  MoveL 2029 to (241.29, 57.14, 41.04) mm, rotated rx 180 ry 0 rz 180 deg; joints [-19.819, 17.595, 47.827, 40.909, 31.181, -36.55]
  Call Extruder(249.57521)
  MoveL 2030 to (241.29, 142.86, 41.03) mm, rotated rx 180 ry 0 rz 180 deg; joints [-28.232, 26.406, 35.284, 48.547, 39.135, -41.289]
  Call Extruder(250.00364)
  MoveL 2031 to (241.27, 143.74, 41.03) mm, rotated rx 180 ry 0 rz -180 deg; joints [-28.313, 26.529, 35.098, 48.584, 39.23, -41.288]
  MoveL 2032 to (241.27, 143.74, 41.03) mm, rotated rx 180 ry 0 rz -180 deg; joints [-28.313, 26.529, 35.098, 48.584, 39.23, -41.288]
  Call Extruder(250.57709)
  MoveL 2033 to (241.22, 144.9, 41.03) mm, rotated rx -180 ry 0 rz 180 deg; joints [-28.421, 26.688, 34.856, 48.637, 39.357, -41.289]
  MoveL 2034 to (241.22, 144.9, 41.03) mm, rotated rx -180 ry 0 rz 180 deg; joints [-28.421, 26.688, 34.856, 48.637, 39.357, -41.289]
  Call Extruder(251.01142)
  MoveL 2035 to (241.18, 145.77, 41.03) mm, rotated rx -180 ry 0 rz 180 deg; joints [-28.503, 26.806, 34.676, 48.678, 39.452, -41.291]
  MoveL 2036 to (241.18, 145.77, 41.03) mm, rotated rx -180 ry 0 rz 180 deg; joints [-28.503, 26.806, 34.676, 48.678, 39.452, -41.291]
  Call Extruder(251.30553)
  MoveL 2037 to (241.13, 146.36, 41.04) mm, rotated rx 180 ry 0 rz 180 deg; joints [-28.559, 26.882, 34.56, 48.708, 39.515, -41.295]
  MoveL 2038 to (241.13, 146.36, 41.04) mm, rotated rx 180 ry 0 rz 180 deg; joints [-28.559, 26.882, 34.56, 48.708, 39.515, -41.295]
  Call Extruder(251.60097)
  MoveL 2039 to (241.09, 146.95, 41.03) mm, rotated rx 180 ry 0 rz 180 deg; joints [-28.615, 26.958, 34.443, 48.737, 39.579, -41.298]
  MoveL 2040 to (241.09, 146.95, 41.03) mm, rotated rx 180 ry 0 rz 180 deg; joints [-28.615, 26.958, 34.443, 48.737, 39.579, -41.298]
  Call Extruder(251.84723)
  MoveL 2041 to (241.04, 147.44, 41.04) mm, rotated rx 180 ry 0 rz -180 deg; joints [-28.662, 27.019, 34.349, 48.762, 39.631, -41.302]
  MoveL 2042 to (241.04, 147.44, 41.04) mm, rotated rx 180 ry 0 rz -180 deg; joints [-28.662, 27.019, 34.349, 48.762, 39.631, -41.302]
  Call Extruder(252.04393)
  MoveL 2043 to (240.99, 147.83, 41.04) mm, rotated rx -180 ry 0 rz 180 deg; joints [-28.7, 27.066, 34.278, 48.784, 39.672, -41.307]
  MoveL 2044 to (240.99, 147.83, 41.04) mm, rotated rx -180 ry 0 rz 180 deg; joints [-28.7, 27.066, 34.278, 48.784, 39.672, -41.307]
  Call Extruder(252.24151)
  MoveL 2045 to (240.95, 148.22, 41.03) mm, rotated rx 180 ry 0 rz 180 deg; joints [-28.737, 27.112, 34.207, 48.806, 39.713, -41.312]
  MoveL 2046 to (240.95, 148.22, 41.03) mm, rotated rx 180 ry 0 rz 180 deg; joints [-28.737, 27.112, 34.207, 48.806, 39.713, -41.312]
  Call Extruder(252.43995)
  MoveL 2047 to (240.9, 148.6, 41.04) mm, rotated rx 180 ry 0 rz 180 deg; joints [-28.774, 27.159, 34.135, 48.827, 39.754, -41.316]
  MoveL 2048 to (240.9, 148.6, 41.04) mm, rotated rx 180 ry 0 rz 180 deg; joints [-28.774, 27.159, 34.135, 48.827, 39.754, -41.316]
  Call Extruder(252.63926)
  MoveL 2049 to (240.86, 148.99, 41.04) mm, rotated rx 180 ry 0 rz -180 deg; joints [-28.812, 27.206, 34.063, 48.848, 39.795, -41.32]
  MoveL 2050 to (240.86, 148.99, 41.04) mm, rotated rx 180 ry 0 rz -180 deg; joints [-28.812, 27.206, 34.063, 48.848, 39.795, -41.32]
  Call Extruder(252.79809)
  MoveL 2051 to (240.81, 149.3, 41.03) mm, rotated rx 180 ry 0 rz 180 deg; joints [-28.842, 27.24, 34.011, 48.867, 39.827, -41.326]
  MoveL 2052 to (240.81, 149.3, 41.03) mm, rotated rx 180 ry 0 rz 180 deg; joints [-28.842, 27.24, 34.011, 48.867, 39.827, -41.326]
  Call Extruder(252.95765)
  MoveL 2053 to (240.76, 149.6, 41.03) mm, rotated rx 180 ry 0 rz 180 deg; joints [-28.872, 27.274, 33.959, 48.886, 39.859, -41.332]
  MoveL 2054 to (240.76, 149.6, 41.03) mm, rotated rx 180 ry 0 rz 180 deg; joints [-28.872, 27.274, 33.959, 48.886, 39.859, -41.332]
  Call Extruder(253.11794)
  MoveL 2055 to (240.71, 149.91, 41.03) mm, rotated rx 180 ry 0 rz 180 deg; joints [-28.902, 27.308, 33.907, 48.905, 39.891, -41.338]
  MoveL 2056 to (240.71, 149.91, 41.03) mm, rotated rx 180 ry 0 rz 180 deg; joints [-28.902, 27.308, 33.907, 48.905, 39.891, -41.338]
  Call Extruder(253.27896)
  MoveL 2057 to (240.66, 150.21, 41.04) mm, rotated rx 180 ry 0 rz 180 deg; joints [-28.932, 27.342, 33.855, 48.924, 39.923, -41.343]
  MoveL 2058 to (240.66, 150.21, 41.04) mm, rotated rx 180 ry 0 rz 180 deg; joints [-28.932, 27.342, 33.855, 48.924, 39.923, -41.343]
  Call Extruder(253.44070)
  MoveL 2059 to (240.61, 150.52, 41.04) mm, rotated rx 180 ry 0 rz -180 deg; joints [-28.962, 27.376, 33.802, 48.942, 39.955, -41.348]
  MoveL 2060 to (240.61, 150.52, 41.04) mm, rotated rx 180 ry 0 rz -180 deg; joints [-28.962, 27.376, 33.802, 48.942, 39.955, -41.348]
  Call Extruder(253.60317)
  MoveL 2061 to (240.57, 150.83, 41.04) mm, rotated rx 180 ry 0 rz 180 deg; joints [-28.993, 27.411, 33.749, 48.961, 39.987, -41.354]
  MoveL 2062 to (240.57, 150.83, 41.04) mm, rotated rx 180 ry 0 rz 180 deg; joints [-28.993, 27.411, 33.749, 48.961, 39.987, -41.354]
  Call Extruder(253.73710)
  MoveL 2063 to (240.52, 151.08, 41.03) mm, rotated rx -180 ry 0 rz 180 deg; joints [-29.017, 27.436, 33.71, 48.977, 40.012, -41.36]
  MoveL 2064 to (240.52, 151.08, 41.03) mm, rotated rx -180 ry 0 rz 180 deg; joints [-29.017, 27.436, 33.71, 48.977, 40.012, -41.36]
  Call Extruder(253.87164)
  MoveL 2065 to (240.47, 151.32, 41.04) mm, rotated rx 180 ry 0 rz 180 deg; joints [-29.043, 27.461, 33.671, 48.994, 40.038, -41.366]
  MoveL 2066 to (240.47, 151.32, 41.04) mm, rotated rx 180 ry 0 rz 180 deg; joints [-29.043, 27.461, 33.671, 48.994, 40.038, -41.366]
  Call Extruder(254.00678)
  MoveL 2067 to (240.42, 151.57, 41.04) mm, rotated rx -180 ry 0 rz -180 deg; joints [-29.067, 27.486, 33.632, 49.011, 40.063, -41.373]
  MoveL 2068 to (240.42, 151.57, 41.04) mm, rotated rx -180 ry 0 rz -180 deg; joints [-29.067, 27.486, 33.632, 49.011, 40.063, -41.373]
  Call Extruder(254.14254)
  MoveL 2069 to (240.37, 151.82, 41.03) mm, rotated rx 180 ry 0 rz 180 deg; joints [-29.092, 27.512, 33.593, 49.028, 40.089, -41.379]
  MoveL 2070 to (240.37, 151.82, 41.03) mm, rotated rx 180 ry 0 rz 180 deg; joints [-29.092, 27.512, 33.593, 49.028, 40.089, -41.379]
  Call Extruder(254.27891)
  MoveL 2071 to (240.32, 152.07, 41.04) mm, rotated rx -180 ry 0 rz 180 deg; joints [-29.117, 27.537, 33.554, 49.045, 40.114, -41.385]
  MoveL 2072 to (240.32, 152.07, 41.04) mm, rotated rx -180 ry 0 rz 180 deg; joints [-29.117, 27.537, 33.554, 49.045, 40.114, -41.385]
  Call Extruder(254.41589)
  MoveL 2073 to (240.27, 152.32, 41.04) mm, rotated rx 180 ry 0 rz 180 deg; joints [-29.142, 27.563, 33.514, 49.061, 40.14, -41.391]
  MoveL 2074 to (240.27, 152.32, 41.04) mm, rotated rx 180 ry 0 rz 180 deg; joints [-29.142, 27.563, 33.514, 49.061, 40.14, -41.391]
  Call Extruder(254.55347)
  MoveL 2075 to (240.22, 152.57, 41.03) mm, rotated rx -180 ry 0 rz 180 deg; joints [-29.167, 27.589, 33.474, 49.078, 40.166, -41.396]
  MoveL 2076 to (240.22, 152.57, 41.03) mm, rotated rx -180 ry 0 rz 180 deg; joints [-29.167, 27.589, 33.474, 49.078, 40.166, -41.396]
  Call Extruder(254.66717)
  MoveL 2077 to (240.17, 152.77, 41.04) mm, rotated rx 180 ry 0 rz 180 deg; joints [-29.188, 27.609, 33.443, 49.092, 40.187, -41.402]
  MoveL 2078 to (240.17, 152.77, 41.04) mm, rotated rx 180 ry 0 rz 180 deg; joints [-29.188, 27.609, 33.443, 49.092, 40.187, -41.402]
  Call Extruder(254.78132)
  MoveL 2079 to (240.13, 152.98, 41.04) mm, rotated rx -180 ry 0 rz 180 deg; joints [-29.209, 27.629, 33.413, 49.106, 40.207, -41.408]
  MoveL 2080 to (240.13, 152.98, 41.04) mm, rotated rx -180 ry 0 rz 180 deg; joints [-29.209, 27.629, 33.413, 49.106, 40.207, -41.408]
  Call Extruder(254.89592)
  MoveL 2081 to (240.08, 153.18, 41.03) mm, rotated rx -180 ry 0 rz -180 deg; joints [-29.229, 27.649, 33.382, 49.121, 40.228, -41.413]
  MoveL 2082 to (240.08, 153.18, 41.03) mm, rotated rx -180 ry 0 rz -180 deg; joints [-29.229, 27.649, 33.382, 49.121, 40.228, -41.413]
  Call Extruder(255.01098)
  MoveL 2083 to (240.04, 153.39, 41.03) mm, rotated rx 180 ry 0 rz 180 deg; joints [-29.25, 27.669, 33.35, 49.135, 40.249, -41.419]
  MoveL 2084 to (240.04, 153.39, 41.03) mm, rotated rx 180 ry 0 rz 180 deg; joints [-29.25, 27.669, 33.35, 49.135, 40.249, -41.419]
  Call Extruder(255.13320)
  MoveL 2085 to (239.98, 153.6, 41.04) mm, rotated rx 180 ry 0 rz 180 deg; joints [-29.272, 27.687, 33.322, 49.151, 40.27, -41.426]
  MoveL 2086 to (239.98, 153.6, 41.04) mm, rotated rx 180 ry 0 rz 180 deg; joints [-29.272, 27.687, 33.322, 49.151, 40.27, -41.426]
  Call Extruder(255.26286)
  MoveL 2087 to (239.92, 153.82, 41.04) mm, rotated rx 180 ry 0 rz 180 deg; joints [-29.296, 27.704, 33.296, 49.171, 40.292, -41.437]
  MoveL 2088 to (239.92, 153.82, 41.04) mm, rotated rx 180 ry 0 rz 180 deg; joints [-29.296, 27.704, 33.296, 49.171, 40.292, -41.437]
  Call Extruder(255.39309)
  MoveL 2089 to (239.85, 154.05, 41.03) mm, rotated rx -180 ry 0 rz -180 deg; joints [-29.319, 27.72, 33.271, 49.19, 40.313, -41.447]
  MoveL 2090 to (239.85, 154.05, 41.03) mm, rotated rx -180 ry 0 rz -180 deg; joints [-29.319, 27.72, 33.271, 49.19, 40.313, -41.447]
  Call Extruder(255.52388)
  MoveL 2091 to (239.78, 154.27, 41.04) mm, rotated rx 180 ry 0 rz 180 deg; joints [-29.343, 27.737, 33.244, 49.209, 40.335, -41.457]
  MoveL 2092 to (239.78, 154.27, 41.04) mm, rotated rx 180 ry 0 rz 180 deg; joints [-29.343, 27.737, 33.244, 49.209, 40.335, -41.457]
  Call Extruder(255.65523)
  MoveL 2093 to (239.71, 154.5, 41.03) mm, rotated rx -180 ry 0 rz 180 deg; joints [-29.366, 27.754, 33.218, 49.228, 40.356, -41.467]
  MoveL 2094 to (239.71, 154.5, 41.03) mm, rotated rx -180 ry 0 rz 180 deg; joints [-29.366, 27.754, 33.218, 49.228, 40.356, -41.467]
  Call Extruder(255.76713)
  MoveL 2095 to (239.65, 154.68, 41.03) mm, rotated rx 180 ry 0 rz 180 deg; joints [-29.386, 27.767, 33.198, 49.245, 40.374, -41.476]
  MoveL 2096 to (239.65, 154.68, 41.03) mm, rotated rx 180 ry 0 rz 180 deg; joints [-29.386, 27.767, 33.198, 49.245, 40.374, -41.476]
  Call Extruder(255.87948)
  MoveL 2097 to (239.59, 154.87, 41.04) mm, rotated rx 180 ry 0 rz 180 deg; joints [-29.406, 27.78, 33.178, 49.261, 40.392, -41.485]
  MoveL 2098 to (239.59, 154.87, 41.04) mm, rotated rx 180 ry 0 rz 180 deg; joints [-29.406, 27.78, 33.178, 49.261, 40.392, -41.485]
  Call Extruder(255.99227)
  MoveL 2099 to (239.53, 155.06, 41.03) mm, rotated rx -180 ry 0 rz 180 deg; joints [-29.426, 27.793, 33.158, 49.278, 40.41, -41.495]
  MoveL 2100 to (239.53, 155.06, 41.03) mm, rotated rx -180 ry 0 rz 180 deg; joints [-29.426, 27.793, 33.158, 49.278, 40.41, -41.495]
  Call Extruder(256.10550)
  MoveL 2101 to (239.47, 155.25, 41.04) mm, rotated rx 180 ry 0 rz 180 deg; joints [-29.446, 27.806, 33.138, 49.295, 40.428, -41.504]
  MoveL 2102 to (239.47, 155.25, 41.04) mm, rotated rx 180 ry 0 rz 180 deg; joints [-29.446, 27.806, 33.138, 49.295, 40.428, -41.504]
  Call Extruder(256.21918)
  MoveL 2103 to (239.41, 155.44, 41.04) mm, rotated rx 180 ry 0 rz 180 deg; joints [-29.466, 27.82, 33.117, 49.312, 40.446, -41.513]
  MoveL 2104 to (239.41, 155.44, 41.04) mm, rotated rx 180 ry 0 rz 180 deg; joints [-29.466, 27.82, 33.117, 49.312, 40.446, -41.513]
  Call Extruder(256.40114)
  MoveL 2105 to (239.29, 155.73, 41.03) mm, rotated rx 180 ry 0 rz -180 deg; joints [-29.499, 27.832, 33.097, 49.343, 40.472, -41.533]
  MoveL 2106 to (239.29, 155.73, 41.03) mm, rotated rx 180 ry 0 rz -180 deg; joints [-29.499, 27.832, 33.097, 49.343, 40.472, -41.533]
  Call Extruder(256.58386)
  MoveL 2107 to (239.16, 156.02, 41.04) mm, rotated rx 180 ry 0 rz 180 deg; joints [-29.531, 27.845, 33.077, 49.374, 40.498, -41.553]
  MoveL 2108 to (239.16, 156.02, 41.04) mm, rotated rx 180 ry 0 rz 180 deg; joints [-29.531, 27.845, 33.077, 49.374, 40.498, -41.553]
  Call Extruder(256.75428)
  MoveL 2109 to (239.05, 156.29, 41.03) mm, rotated rx -180 ry 0 rz 180 deg; joints [-29.561, 27.857, 33.06, 49.403, 40.522, -41.572]
  MoveL 2110 to (239.05, 156.29, 41.03) mm, rotated rx -180 ry 0 rz 180 deg; joints [-29.561, 27.857, 33.06, 49.403, 40.522, -41.572]
  Call Extruder(256.91229)
  MoveL 2111 to (238.94, 156.54, 41.04) mm, rotated rx 180 ry 0 rz 180 deg; joints [-29.589, 27.867, 33.044, 49.43, 40.544, -41.59]
  MoveL 2112 to (238.94, 156.54, 41.04) mm, rotated rx 180 ry 0 rz 180 deg; joints [-29.589, 27.867, 33.044, 49.43, 40.544, -41.59]
  Call Extruder(257.07091)
  MoveL 2113 to (238.84, 156.79, 41.04) mm, rotated rx 180 ry 0 rz 180 deg; joints [-29.617, 27.877, 33.028, 49.457, 40.566, -41.608]
  MoveL 2114 to (238.84, 156.79, 41.04) mm, rotated rx 180 ry 0 rz 180 deg; joints [-29.617, 27.877, 33.028, 49.457, 40.566, -41.608]
  Call Extruder(257.27708)
  MoveL 2115 to (238.66, 157.09, 41.04) mm, rotated rx -180 ry 0 rz 180 deg; joints [-29.653, 27.876, 33.029, 49.499, 40.59, -41.64]
  MoveL 2116 to (238.66, 157.09, 41.04) mm, rotated rx -180 ry 0 rz 180 deg; joints [-29.653, 27.876, 33.029, 49.499, 40.59, -41.64]
  Call Extruder(257.48403)
  MoveL 2117 to (238.49, 157.4, 41.04) mm, rotated rx 180 ry 0 rz 180 deg; joints [-29.689, 27.875, 33.031, 49.541, 40.614, -41.672]
  MoveL 2118 to (238.49, 157.4, 41.04) mm, rotated rx 180 ry 0 rz 180 deg; joints [-29.689, 27.875, 33.031, 49.541, 40.614, -41.672]
  Call Extruder(257.69175)
  MoveL 2119 to (238.31, 157.7, 41.04) mm, rotated rx 180 ry 0 rz 180 deg; joints [-29.725, 27.875, 33.031, 49.582, 40.638, -41.704]
  MoveL 2120 to (238.31, 157.7, 41.04) mm, rotated rx 180 ry 0 rz 180 deg; joints [-29.725, 27.875, 33.031, 49.582, 40.638, -41.704]
  Call Extruder(257.90025)
  MoveL 2121 to (238.13, 158.01, 41.04) mm, rotated rx -180 ry 0 rz 180 deg; joints [-29.761, 27.874, 33.032, 49.624, 40.662, -41.736]
  MoveL 2122 to (238.13, 158.01, 41.04) mm, rotated rx -180 ry 0 rz 180 deg; joints [-29.761, 27.874, 33.032, 49.624, 40.662, -41.736]
  Call Extruder(258.07978)
  MoveL 2123 to (237.96, 158.25, 41.04) mm, rotated rx -180 ry 0 rz 180 deg; joints [-29.792, 27.864, 33.049, 49.665, 40.678, -41.769]
  MoveL 2124 to (237.96, 158.25, 41.04) mm, rotated rx -180 ry 0 rz 180 deg; joints [-29.792, 27.864, 33.049, 49.665, 40.678, -41.769]
  Call Extruder(258.41320)
  MoveL 2125 to (237.63, 158.7, 41.03) mm, rotated rx 180 ry 0 rz 180 deg; joints [-29.849, 27.844, 33.08, 49.74, 40.709, -41.832]
  MoveL 2126 to (237.63, 158.7, 41.03) mm, rotated rx 180 ry 0 rz 180 deg; joints [-29.849, 27.844, 33.08, 49.74, 40.709, -41.832]
  Call Extruder(258.74780)
  MoveL 2127 to (237.3, 159.15, 41.04) mm, rotated rx 180 ry 0 rz 180 deg; joints [-29.907, 27.824, 33.11, 49.815, 40.741, -41.894]
  Call Extruder(259.57575)
  MoveL 2128 to (236.39, 160.19, 41.03) mm, rotated rx 180 ry 0 rz 180 deg; joints [-30.046, 27.733, 33.251, 50.018, 40.802, -42.072]
  Call Extruder(260.40368)
  MoveL 2129 to (235.35, 161.1, 41.03) mm, rotated rx -180 ry 0 rz 180 deg; joints [-30.182, 27.588, 33.475, 50.241, 40.842, -42.281]
  Call Extruder(260.57099)
  MoveL 2130 to (235.13, 161.27, 41.04) mm, rotated rx 180 ry 0 rz 180 deg; joints [-30.208, 27.551, 33.532, 50.289, 40.847, -42.328]
  MoveL 2131 to (235.13, 161.27, 41.04) mm, rotated rx 180 ry 0 rz 180 deg; joints [-30.208, 27.551, 33.532, 50.289, 40.847, -42.328]
  Call Extruder(260.90442)
  MoveL 2132 to (234.68, 161.59, 41.04) mm, rotated rx 180 ry 0 rz -180 deg; joints [-30.261, 27.478, 33.646, 50.384, 40.857, -42.42]
  MoveL 2133 to (234.68, 161.59, 41.04) mm, rotated rx 180 ry 0 rz -180 deg; joints [-30.261, 27.478, 33.646, 50.384, 40.857, -42.42]
  Call Extruder(261.23666)
  MoveL 2134 to (234.23, 161.92, 41.04) mm, rotated rx 180 ry 0 rz 180 deg; joints [-30.314, 27.404, 33.758, 50.479, 40.868, -42.511]
  MoveL 2135 to (234.23, 161.92, 41.04) mm, rotated rx 180 ry 0 rz 180 deg; joints [-30.314, 27.404, 33.758, 50.479, 40.868, -42.511]
  Call Extruder(261.35431)
  MoveL 2136 to (234.05, 162.02, 41.04) mm, rotated rx -180 ry 0 rz 180 deg; joints [-30.331, 27.373, 33.807, 50.514, 40.869, -42.547]
  MoveL 2137 to (234.05, 162.02, 41.04) mm, rotated rx -180 ry 0 rz 180 deg; joints [-30.331, 27.373, 33.807, 50.514, 40.869, -42.547]
  Call Extruder(261.56204)
  MoveL 2138 to (233.75, 162.2, 41.04) mm, rotated rx -180 ry 0 rz 180 deg; joints [-30.363, 27.316, 33.894, 50.577, 40.871, -42.609]
  MoveL 2139 to (233.75, 162.2, 41.04) mm, rotated rx -180 ry 0 rz 180 deg; joints [-30.363, 27.316, 33.894, 50.577, 40.871, -42.609]
  Call Extruder(261.76899)
  MoveL 2140 to (233.45, 162.37, 41.04) mm, rotated rx -180 ry 0 rz 180 deg; joints [-30.394, 27.26, 33.98, 50.639, 40.873, -42.672]
  MoveL 2141 to (233.45, 162.37, 41.04) mm, rotated rx -180 ry 0 rz 180 deg; joints [-30.394, 27.26, 33.98, 50.639, 40.873, -42.672]
  Call Extruder(261.97516)
  MoveL 2142 to (233.14, 162.55, 41.03) mm, rotated rx 180 ry 0 rz 180 deg; joints [-30.426, 27.204, 34.066, 50.701, 40.875, -42.734]
  MoveL 2143 to (233.14, 162.55, 41.03) mm, rotated rx 180 ry 0 rz 180 deg; joints [-30.426, 27.204, 34.066, 50.701, 40.875, -42.734]
  Call Extruder(262.15683)
  MoveL 2144 to (232.87, 162.69, 41.04) mm, rotated rx 180 ry 0 rz 180 deg; joints [-30.453, 27.151, 34.148, 50.758, 40.876, -42.791]
  MoveL 2145 to (232.87, 162.69, 41.04) mm, rotated rx 180 ry 0 rz 180 deg; joints [-30.453, 27.151, 34.148, 50.758, 40.876, -42.791]
  Call Extruder(262.31480)
  MoveL 2146 to (232.62, 162.8, 41.04) mm, rotated rx 180 ry 0 rz 180 deg; joints [-30.476, 27.1, 34.227, 50.807, 40.874, -42.842]
  MoveL 2147 to (232.62, 162.8, 41.04) mm, rotated rx 180 ry 0 rz 180 deg; joints [-30.476, 27.1, 34.227, 50.807, 40.874, -42.842]
  Call Extruder(262.47217)
  MoveL 2148 to (232.37, 162.91, 41.04) mm, rotated rx 180 ry 0 rz 180 deg; joints [-30.498, 27.048, 34.305, 50.857, 40.872, -42.894]
  MoveL 2149 to (232.37, 162.91, 41.04) mm, rotated rx 180 ry 0 rz 180 deg; joints [-30.498, 27.048, 34.305, 50.857, 40.872, -42.894]
  Call Extruder(262.65491)
  MoveL 2150 to (232.07, 163.02, 41.04) mm, rotated rx -180 ry 0 rz 180 deg; joints [-30.524, 26.988, 34.398, 50.915, 40.869, -42.954]
  MoveL 2151 to (232.07, 163.02, 41.04) mm, rotated rx -180 ry 0 rz 180 deg; joints [-30.524, 26.988, 34.398, 50.915, 40.869, -42.954]
  Call Extruder(262.83690)
  MoveL 2152 to (231.78, 163.15, 41.03) mm, rotated rx -180 ry 0 rz 180 deg; joints [-30.551, 26.928, 34.49, 50.973, 40.867, -43.014]
  MoveL 2153 to (231.78, 163.15, 41.03) mm, rotated rx -180 ry 0 rz 180 deg; joints [-30.551, 26.928, 34.49, 50.973, 40.867, -43.014]
  Call Extruder(262.98424)
  MoveL 2154 to (231.54, 163.24, 41.04) mm, rotated rx 180 ry 0 rz 180 deg; joints [-30.571, 26.877, 34.567, 51.02, 40.865, -43.063]
  MoveL 2155 to (231.54, 163.24, 41.04) mm, rotated rx 180 ry 0 rz 180 deg; joints [-30.571, 26.877, 34.567, 51.02, 40.865, -43.063]
  Call Extruder(263.09746)
  MoveL 2156 to (231.35, 163.3, 41.03) mm, rotated rx 180 ry 0 rz 180 deg; joints [-30.587, 26.836, 34.63, 51.057, 40.861, -43.102]
  MoveL 2157 to (231.35, 163.3, 41.03) mm, rotated rx 180 ry 0 rz 180 deg; joints [-30.587, 26.836, 34.63, 51.057, 40.861, -43.102]
  Call Extruder(263.21024)
  MoveL 2158 to (231.17, 163.36, 41.03) mm, rotated rx 180 ry 0 rz 180 deg; joints [-30.602, 26.795, 34.693, 51.094, 40.858, -43.141]
  MoveL 2159 to (231.17, 163.36, 41.03) mm, rotated rx 180 ry 0 rz 180 deg; joints [-30.602, 26.795, 34.693, 51.094, 40.858, -43.141]
  Call Extruder(263.32257)
  MoveL 2160 to (230.98, 163.42, 41.04) mm, rotated rx 180 ry 0 rz 180 deg; joints [-30.618, 26.753, 34.756, 51.13, 40.855, -43.179]
  MoveL 2161 to (230.98, 163.42, 41.04) mm, rotated rx 180 ry 0 rz 180 deg; joints [-30.618, 26.753, 34.756, 51.13, 40.855, -43.179]
  Call Extruder(263.43446)
  MoveL 2162 to (230.79, 163.48, 41.04) mm, rotated rx 180 ry 0 rz 180 deg; joints [-30.633, 26.712, 34.818, 51.167, 40.852, -43.218]
  MoveL 2163 to (230.79, 163.48, 41.04) mm, rotated rx 180 ry 0 rz 180 deg; joints [-30.633, 26.712, 34.818, 51.167, 40.852, -43.218]
  Call Extruder(263.55586)
  MoveL 2164 to (230.58, 163.55, 41.04) mm, rotated rx 180 ry 0 rz 180 deg; joints [-30.65, 26.667, 34.887, 51.207, 40.849, -43.26]
  MoveL 2165 to (230.58, 163.55, 41.04) mm, rotated rx 180 ry 0 rz 180 deg; joints [-30.65, 26.667, 34.887, 51.207, 40.849, -43.26]
  Call Extruder(263.68667)
  MoveL 2166 to (230.36, 163.61, 41.03) mm, rotated rx -180 ry 0 rz 180 deg; joints [-30.668, 26.618, 34.962, 51.25, 40.845, -43.306]
  MoveL 2167 to (230.36, 163.61, 41.03) mm, rotated rx -180 ry 0 rz 180 deg; joints [-30.668, 26.618, 34.962, 51.25, 40.845, -43.306]
  Call Extruder(263.81692)
  MoveL 2168 to (230.14, 163.68, 41.03) mm, rotated rx 180 ry 0 rz 180 deg; joints [-30.685, 26.569, 35.036, 51.293, 40.842, -43.351]
  MoveL 2169 to (230.14, 163.68, 41.03) mm, rotated rx 180 ry 0 rz 180 deg; joints [-30.685, 26.569, 35.036, 51.293, 40.842, -43.351]
  Call Extruder(263.94661)
  MoveL 2170 to (229.91, 163.75, 41.04) mm, rotated rx 180 ry 0 rz 180 deg; joints [-30.703, 26.521, 35.11, 51.335, 40.838, -43.397]
  MoveL 2171 to (229.91, 163.75, 41.04) mm, rotated rx 180 ry 0 rz 180 deg; joints [-30.703, 26.521, 35.11, 51.335, 40.838, -43.397]
  Call Extruder(264.07572)
  MoveL 2172 to (229.69, 163.82, 41.03) mm, rotated rx -180 ry 0 rz 180 deg; joints [-30.721, 26.472, 35.185, 51.378, 40.834, -43.442]
  MoveL 2173 to (229.69, 163.82, 41.03) mm, rotated rx -180 ry 0 rz 180 deg; joints [-30.721, 26.472, 35.185, 51.378, 40.834, -43.442]
  Call Extruder(264.19080)
  MoveL 2174 to (229.48, 163.86, 41.04) mm, rotated rx 180 ry 0 rz 180 deg; joints [-30.736, 26.425, 35.256, 51.417, 40.83, -43.483]
  MoveL 2175 to (229.48, 163.86, 41.04) mm, rotated rx 180 ry 0 rz 180 deg; joints [-30.736, 26.425, 35.256, 51.417, 40.83, -43.483]
  Call Extruder(264.30542)
  MoveL 2176 to (229.28, 163.91, 41.04) mm, rotated rx 180 ry 0 rz 180 deg; joints [-30.751, 26.378, 35.327, 51.455, 40.825, -43.525]
  MoveL 2177 to (229.28, 163.91, 41.04) mm, rotated rx 180 ry 0 rz 180 deg; joints [-30.751, 26.378, 35.327, 51.455, 40.825, -43.525]
  Call Extruder(264.41959)
  MoveL 2178 to (229.08, 163.95, 41.04) mm, rotated rx 180 ry 0 rz -180 deg; joints [-30.766, 26.331, 35.398, 51.493, 40.82, -43.566]
  MoveL 2179 to (229.08, 163.95, 41.04) mm, rotated rx 180 ry 0 rz -180 deg; joints [-30.766, 26.331, 35.398, 51.493, 40.82, -43.566]
  Call Extruder(264.53331)
  MoveL 2180 to (228.87, 164, 41.03) mm, rotated rx 180 ry 0 rz 180 deg; joints [-30.781, 26.284, 35.468, 51.532, 40.815, -43.607]
  MoveL 2181 to (228.87, 164, 41.03) mm, rotated rx 180 ry 0 rz 180 deg; joints [-30.781, 26.284, 35.468, 51.532, 40.815, -43.607]
  Call Extruder(264.65873)
  MoveL 2182 to (228.65, 164.04, 41.03) mm, rotated rx 180 ry 0 rz 180 deg; joints [-30.797, 26.233, 35.547, 51.574, 40.81, -43.653]
  MoveL 2183 to (228.65, 164.04, 41.03) mm, rotated rx 180 ry 0 rz 180 deg; joints [-30.797, 26.233, 35.547, 51.574, 40.81, -43.653]
  Call Extruder(264.79570)
  MoveL 2184 to (228.4, 164.09, 41.04) mm, rotated rx 180 ry 0 rz -180 deg; joints [-30.815, 26.176, 35.633, 51.62, 40.804, -43.703]
  MoveL 2185 to (228.4, 164.09, 41.04) mm, rotated rx 180 ry 0 rz -180 deg; joints [-30.815, 26.176, 35.633, 51.62, 40.804, -43.703]
  Call Extruder(264.93207)
  MoveL 2186 to (228.15, 164.14, 41.04) mm, rotated rx 180 ry 0 rz 180 deg; joints [-30.832, 26.118, 35.72, 51.666, 40.798, -43.753]
  MoveL 2187 to (228.15, 164.14, 41.04) mm, rotated rx 180 ry 0 rz 180 deg; joints [-30.832, 26.118, 35.72, 51.666, 40.798, -43.753]
  Call Extruder(265.06783)
  MoveL 2188 to (227.9, 164.19, 41.04) mm, rotated rx 180 ry 0 rz -180 deg; joints [-30.85, 26.061, 35.806, 51.712, 40.792, -43.803]
  MoveL 2189 to (227.9, 164.19, 41.04) mm, rotated rx 180 ry 0 rz -180 deg; joints [-30.85, 26.061, 35.806, 51.712, 40.792, -43.803]
  Call Extruder(265.20298)
  MoveL 2190 to (227.65, 164.24, 41.03) mm, rotated rx 180 ry 0 rz 180 deg; joints [-30.868, 26.005, 35.891, 51.758, 40.787, -43.852]
  MoveL 2191 to (227.65, 164.24, 41.03) mm, rotated rx 180 ry 0 rz 180 deg; joints [-30.868, 26.005, 35.891, 51.758, 40.787, -43.852]
  Call Extruder(265.33751)
  MoveL 2192 to (227.4, 164.29, 41.04) mm, rotated rx 180 ry 0 rz 180 deg; joints [-30.886, 25.948, 35.977, 51.804, 40.781, -43.901]
  MoveL 2193 to (227.4, 164.29, 41.04) mm, rotated rx 180 ry 0 rz 180 deg; joints [-30.886, 25.948, 35.977, 51.804, 40.781, -43.901]
  Call Extruder(265.47144)
  MoveL 2194 to (227.15, 164.34, 41.04) mm, rotated rx -180 ry 0 rz -180 deg; joints [-30.903, 25.892, 36.061, 51.849, 40.776, -43.951]
  MoveL 2195 to (227.15, 164.34, 41.04) mm, rotated rx -180 ry 0 rz -180 deg; joints [-30.903, 25.892, 36.061, 51.849, 40.776, -43.951]
  Call Extruder(265.61931)
  MoveL 2196 to (226.87, 164.39, 41.03) mm, rotated rx -180 ry 0 rz 180 deg; joints [-30.923, 25.828, 36.157, 51.9, 40.769, -44.005]
  MoveL 2197 to (226.87, 164.39, 41.03) mm, rotated rx -180 ry 0 rz 180 deg; joints [-30.923, 25.828, 36.157, 51.9, 40.769, -44.005]
  Call Extruder(265.78105)
  MoveL 2198 to (226.57, 164.44, 41.04) mm, rotated rx 180 ry 0 rz 180 deg; joints [-30.943, 25.758, 36.263, 51.955, 40.762, -44.065]
  MoveL 2199 to (226.57, 164.44, 41.04) mm, rotated rx 180 ry 0 rz 180 deg; joints [-30.943, 25.758, 36.263, 51.955, 40.762, -44.065]
  Call Extruder(265.94206)
  MoveL 2200 to (226.26, 164.49, 41.04) mm, rotated rx 180 ry 0 rz 180 deg; joints [-30.964, 25.688, 36.368, 52.01, 40.755, -44.125]
  MoveL 2201 to (226.26, 164.49, 41.04) mm, rotated rx 180 ry 0 rz 180 deg; joints [-30.964, 25.688, 36.368, 52.01, 40.755, -44.125]
  Call Extruder(266.10234)
  MoveL 2202 to (225.96, 164.53, 41.03) mm, rotated rx -180 ry 0 rz 180 deg; joints [-30.985, 25.618, 36.473, 52.065, 40.748, -44.185]
  MoveL 2203 to (225.96, 164.53, 41.03) mm, rotated rx -180 ry 0 rz 180 deg; joints [-30.985, 25.618, 36.473, 52.065, 40.748, -44.185]
  Call Extruder(266.26190)
  MoveL 2204 to (225.65, 164.58, 41.04) mm, rotated rx 180 ry 0 rz 180 deg; joints [-31.006, 25.548, 36.578, 52.12, 40.741, -44.244]
  MoveL 2205 to (225.65, 164.58, 41.04) mm, rotated rx 180 ry 0 rz 180 deg; joints [-31.006, 25.548, 36.578, 52.12, 40.741, -44.244]
  Call Extruder(266.42073)
  MoveL 2206 to (225.34, 164.63, 41.03) mm, rotated rx 180 ry 0 rz -180 deg; joints [-31.027, 25.479, 36.682, 52.174, 40.734, -44.303]
  MoveL 2207 to (225.34, 164.63, 41.03) mm, rotated rx 180 ry 0 rz -180 deg; joints [-31.027, 25.479, 36.682, 52.174, 40.734, -44.303]
  Call Extruder(266.59940)
  MoveL 2208 to (225, 164.68, 41.04) mm, rotated rx 180 ry 0 rz -180 deg; joints [-31.049, 25.399, 36.801, 52.235, 40.726, -44.37]
  MoveL 2209 to (225, 164.68, 41.04) mm, rotated rx 180 ry 0 rz -180 deg; joints [-31.049, 25.399, 36.801, 52.235, 40.726, -44.37]
  Call Extruder(266.79784)
  MoveL 2210 to (224.61, 164.73, 41.04) mm, rotated rx -180 ry 0 rz -180 deg; joints [-31.074, 25.31, 36.934, 52.303, 40.716, -44.444]
  MoveL 2211 to (224.61, 164.73, 41.04) mm, rotated rx -180 ry 0 rz -180 deg; joints [-31.074, 25.31, 36.934, 52.303, 40.716, -44.444]
  Call Extruder(266.99542)
  MoveL 2212 to (224.22, 164.77, 41.03) mm, rotated rx 180 ry 0 rz 180 deg; joints [-31.1, 25.22, 37.067, 52.371, 40.707, -44.518]
  MoveL 2213 to (224.22, 164.77, 41.03) mm, rotated rx 180 ry 0 rz 180 deg; joints [-31.1, 25.22, 37.067, 52.371, 40.707, -44.518]
  Call Extruder(267.19212)
  MoveL 2214 to (223.84, 164.82, 41.04) mm, rotated rx 180 ry 0 rz 180 deg; joints [-31.125, 25.132, 37.199, 52.439, 40.698, -44.592]
  MoveL 2215 to (223.84, 164.82, 41.04) mm, rotated rx 180 ry 0 rz 180 deg; joints [-31.125, 25.132, 37.199, 52.439, 40.698, -44.592]
  Call Extruder(267.38796)
  MoveL 2216 to (223.45, 164.86, 41.03) mm, rotated rx 180 ry 0 rz 180 deg; joints [-31.15, 25.043, 37.331, 52.506, 40.69, -44.665]
  MoveL 2217 to (223.45, 164.86, 41.03) mm, rotated rx 180 ry 0 rz 180 deg; joints [-31.15, 25.043, 37.331, 52.506, 40.69, -44.665]
  Call Extruder(267.68332)
  MoveL 2218 to (222.86, 164.91, 41.04) mm, rotated rx 180 ry 0 rz 180 deg; joints [-31.186, 24.907, 37.534, 52.607, 40.675, -44.776]
  MoveL 2219 to (222.86, 164.91, 41.04) mm, rotated rx 180 ry 0 rz 180 deg; joints [-31.186, 24.907, 37.534, 52.607, 40.675, -44.776]
  Call Extruder(267.97734)
  MoveL 2220 to (222.27, 164.95, 41.04) mm, rotated rx 180 ry 0 rz 180 deg; joints [-31.222, 24.771, 37.736, 52.707, 40.66, -44.886]
  MoveL 2221 to (222.27, 164.95, 41.04) mm, rotated rx 180 ry 0 rz 180 deg; joints [-31.222, 24.771, 37.736, 52.707, 40.66, -44.886]
  Call Extruder(268.27004)
  MoveL 2222 to (221.68, 165, 41.04) mm, rotated rx 180 ry 0 rz 180 deg; joints [-31.258, 24.636, 37.935, 52.806, 40.647, -44.995]
  MoveL 2223 to (221.68, 165, 41.04) mm, rotated rx 180 ry 0 rz 180 deg; joints [-31.258, 24.636, 37.935, 52.806, 40.647, -44.995]
  Call Extruder(268.84349)
  MoveL 2224 to (220.52, 165.05, 41.04) mm, rotated rx 180 ry 0 rz 180 deg; joints [-31.326, 24.366, 38.334, 52.999, 40.617, -45.208]
  MoveL 2225 to (220.52, 165.05, 41.04) mm, rotated rx 180 ry 0 rz 180 deg; joints [-31.326, 24.366, 38.334, 52.999, 40.617, -45.208]
  Call Extruder(269.55750)
  MoveL 2226 to (219.06, 165.09, 41.03) mm, rotated rx 180 ry 0 rz 180 deg; joints [-31.409, 24.03, 38.827, 53.236, 40.582, -45.47]
  Call Extruder(386.40424)
  MoveL 2227 to (-19.06, 165.09, 41.04) mm, rotated rx 180 ry 0 rz 180 deg; joints [-51.475, -8.459, 76.118, 73.163, 54.823, -62.287]
  Call Extruder(386.83284)
  MoveL 2228 to (-19.94, 165.07, 41.04) mm, rotated rx -180 ry 0 rz 180 deg; joints [-51.582, -8.539, 76.186, 73.215, 54.921, -62.307]
  MoveL 2229 to (-19.94, 165.07, 41.04) mm, rotated rx -180 ry 0 rz 180 deg; joints [-51.582, -8.539, 76.186, 73.215, 54.921, -62.307]
  Call Extruder(387.40629)
  MoveL 2230 to (-21.1, 165.03, 41.04) mm, rotated rx 180 ry 0 rz 180 deg; joints [-51.722, -8.648, 76.277, 73.283, 55.051, -62.332]
  MoveL 2231 to (-21.1, 165.03, 41.04) mm, rotated rx 180 ry 0 rz 180 deg; joints [-51.722, -8.648, 76.277, 73.283, 55.051, -62.332]
  Call Extruder(387.84059)
  MoveL 2232 to (-21.97, 164.98, 41.04) mm, rotated rx 180 ry 0 rz 180 deg; joints [-51.827, -8.731, 76.347, 73.333, 55.147, -62.351]
  MoveL 2233 to (-21.97, 164.98, 41.04) mm, rotated rx 180 ry 0 rz 180 deg; joints [-51.827, -8.731, 76.347, 73.333, 55.147, -62.351]
  Call Extruder(388.13462)
  MoveL 2234 to (-22.56, 164.93, 41.04) mm, rotated rx 180 ry 0 rz -180 deg; joints [-51.897, -8.788, 76.395, 73.366, 55.212, -62.362]
  MoveL 2235 to (-22.56, 164.93, 41.04) mm, rotated rx 180 ry 0 rz -180 deg; joints [-51.897, -8.788, 76.395, 73.366, 55.212, -62.362]
  Call Extruder(388.42998)
  MoveL 2236 to (-23.15, 164.89, 41.04) mm, rotated rx 180 ry 0 rz 180 deg; joints [-51.966, -8.846, 76.443, 73.399, 55.276, -62.374]
  MoveL 2237 to (-23.15, 164.89, 41.04) mm, rotated rx 180 ry 0 rz 180 deg; joints [-51.966, -8.846, 76.443, 73.399, 55.276, -62.374]
  Call Extruder(388.67619)
  MoveL 2238 to (-23.64, 164.84, 41.04) mm, rotated rx 180 ry 0 rz 180 deg; joints [-52.023, -8.894, 76.483, 73.426, 55.328, -62.382]
  MoveL 2239 to (-23.64, 164.84, 41.04) mm, rotated rx 180 ry 0 rz 180 deg; joints [-52.023, -8.894, 76.483, 73.426, 55.328, -62.382]
  Call Extruder(388.87290)
  MoveL 2240 to (-24.03, 164.79, 41.04) mm, rotated rx -180 ry 0 rz 180 deg; joints [-52.067, -8.933, 76.516, 73.447, 55.37, -62.389]
  MoveL 2241 to (-24.03, 164.79, 41.04) mm, rotated rx -180 ry 0 rz 180 deg; joints [-52.067, -8.933, 76.516, 73.447, 55.37, -62.389]
  Call Extruder(389.07047)
  MoveL 2242 to (-24.42, 164.75, 41.04) mm, rotated rx 180 ry 0 rz 180 deg; joints [-52.112, -8.973, 76.548, 73.467, 55.411, -62.396]
  MoveL 2243 to (-24.42, 164.75, 41.04) mm, rotated rx 180 ry 0 rz 180 deg; joints [-52.112, -8.973, 76.548, 73.467, 55.411, -62.396]
  Call Extruder(389.26891)
  MoveL 2244 to (-24.8, 164.7, 41.04) mm, rotated rx 180 ry 0 rz 180 deg; joints [-52.156, -9.012, 76.581, 73.488, 55.452, -62.402]
  MoveL 2245 to (-24.8, 164.7, 41.04) mm, rotated rx 180 ry 0 rz 180 deg; joints [-52.156, -9.012, 76.581, 73.488, 55.452, -62.402]
  Call Extruder(389.46822)
  MoveL 2246 to (-25.19, 164.66, 41.04) mm, rotated rx 180 ry 0 rz 180 deg; joints [-52.2, -9.051, 76.614, 73.509, 55.493, -62.409]
  MoveL 2247 to (-25.19, 164.66, 41.04) mm, rotated rx 180 ry 0 rz 180 deg; joints [-52.2, -9.051, 76.614, 73.509, 55.493, -62.409]
  Call Extruder(389.62706)
  MoveL 2248 to (-25.5, 164.61, 41.04) mm, rotated rx -180 ry 0 rz 180 deg; joints [-52.235, -9.083, 76.64, 73.524, 55.525, -62.413]
  MoveL 2249 to (-25.5, 164.61, 41.04) mm, rotated rx -180 ry 0 rz 180 deg; joints [-52.235, -9.083, 76.64, 73.524, 55.525, -62.413]
  Call Extruder(389.78661)
  MoveL 2250 to (-25.8, 164.56, 41.04) mm, rotated rx -180 ry 0 rz 180 deg; joints [-52.269, -9.116, 76.667, 73.54, 55.557, -62.418]
  MoveL 2251 to (-25.8, 164.56, 41.04) mm, rotated rx -180 ry 0 rz 180 deg; joints [-52.269, -9.116, 76.667, 73.54, 55.557, -62.418]
  Call Extruder(389.94690)
  MoveL 2252 to (-26.11, 164.51, 41.04) mm, rotated rx -180 ry 0 rz 180 deg; joints [-52.303, -9.148, 76.694, 73.555, 55.588, -62.422]
  MoveL 2253 to (-26.11, 164.51, 41.04) mm, rotated rx -180 ry 0 rz 180 deg; joints [-52.303, -9.148, 76.694, 73.555, 55.588, -62.422]
  Call Extruder(390.10792)
  MoveL 2254 to (-26.41, 164.46, 41.04) mm, rotated rx 180 ry 0 rz 180 deg; joints [-52.337, -9.18, 76.721, 73.571, 55.62, -62.426]
  MoveL 2255 to (-26.41, 164.46, 41.04) mm, rotated rx 180 ry 0 rz 180 deg; joints [-52.337, -9.18, 76.721, 73.571, 55.62, -62.426]
  Call Extruder(390.26966)
  MoveL 2256 to (-26.72, 164.41, 41.04) mm, rotated rx 180 ry 0 rz 180 deg; joints [-52.371, -9.212, 76.747, 73.586, 55.652, -62.431]
  MoveL 2257 to (-26.72, 164.41, 41.04) mm, rotated rx 180 ry 0 rz 180 deg; joints [-52.371, -9.212, 76.747, 73.586, 55.652, -62.431]
  Call Extruder(390.43213)
  MoveL 2258 to (-27.03, 164.37, 41.04) mm, rotated rx 180 ry 0 rz -180 deg; joints [-52.405, -9.244, 76.774, 73.602, 55.684, -62.435]
  MoveL 2259 to (-27.03, 164.37, 41.04) mm, rotated rx 180 ry 0 rz -180 deg; joints [-52.405, -9.244, 76.774, 73.602, 55.684, -62.435]
  Call Extruder(390.56606)
  MoveL 2260 to (-27.27, 164.32, 41.04) mm, rotated rx 180 ry 0 rz 180 deg; joints [-52.432, -9.271, 76.796, 73.614, 55.709, -62.438]
  MoveL 2261 to (-27.27, 164.32, 41.04) mm, rotated rx 180 ry 0 rz 180 deg; joints [-52.432, -9.271, 76.796, 73.614, 55.709, -62.438]
  Call Extruder(390.70059)
  MoveL 2262 to (-27.52, 164.27, 41.04) mm, rotated rx -180 ry 0 rz 180 deg; joints [-52.459, -9.299, 76.819, 73.626, 55.734, -62.441]
  MoveL 2263 to (-27.52, 164.27, 41.04) mm, rotated rx -180 ry 0 rz 180 deg; joints [-52.459, -9.299, 76.819, 73.626, 55.734, -62.441]
  Call Extruder(390.83574)
  MoveL 2264 to (-27.77, 164.22, 41.04) mm, rotated rx 180 ry 0 rz 180 deg; joints [-52.486, -9.326, 76.841, 73.638, 55.76, -62.444]
  MoveL 2265 to (-27.77, 164.22, 41.04) mm, rotated rx 180 ry 0 rz 180 deg; joints [-52.486, -9.326, 76.841, 73.638, 55.76, -62.444]
  Call Extruder(390.97150)
  MoveL 2266 to (-28.02, 164.17, 41.04) mm, rotated rx -180 ry 0 rz -180 deg; joints [-52.513, -9.353, 76.864, 73.65, 55.785, -62.447]
  MoveL 2267 to (-28.02, 164.17, 41.04) mm, rotated rx -180 ry 0 rz -180 deg; joints [-52.513, -9.353, 76.864, 73.65, 55.785, -62.447]
  Call Extruder(391.10786)
  MoveL 2268 to (-28.27, 164.12, 41.04) mm, rotated rx 180 ry 0 rz 180 deg; joints [-52.54, -9.38, 76.886, 73.662, 55.81, -62.45]
  MoveL 2269 to (-28.27, 164.12, 41.04) mm, rotated rx 180 ry 0 rz 180 deg; joints [-52.54, -9.38, 76.886, 73.662, 55.81, -62.45]
  Call Extruder(391.24484)
  MoveL 2270 to (-28.52, 164.07, 41.04) mm, rotated rx 180 ry 0 rz 180 deg; joints [-52.567, -9.408, 76.909, 73.674, 55.835, -62.453]
  MoveL 2271 to (-28.52, 164.07, 41.04) mm, rotated rx 180 ry 0 rz 180 deg; joints [-52.567, -9.408, 76.909, 73.674, 55.835, -62.453]
  Call Extruder(391.38243)
  MoveL 2272 to (-28.77, 164.02, 41.04) mm, rotated rx 180 ry 0 rz 180 deg; joints [-52.594, -9.435, 76.931, 73.686, 55.861, -62.456]
  MoveL 2273 to (-28.77, 164.02, 41.04) mm, rotated rx 180 ry 0 rz 180 deg; joints [-52.594, -9.435, 76.931, 73.686, 55.861, -62.456]
  Call Extruder(391.49614)
  MoveL 2274 to (-28.97, 163.97, 41.04) mm, rotated rx 180 ry 0 rz 180 deg; joints [-52.616, -9.458, 76.95, 73.695, 55.881, -62.458]
  MoveL 2275 to (-28.97, 163.97, 41.04) mm, rotated rx 180 ry 0 rz 180 deg; joints [-52.616, -9.458, 76.95, 73.695, 55.881, -62.458]
  Call Extruder(391.61031)
  MoveL 2276 to (-29.18, 163.93, 41.04) mm, rotated rx -180 ry 0 rz -180 deg; joints [-52.638, -9.48, 76.969, 73.705, 55.902, -62.46]
  MoveL 2277 to (-29.18, 163.93, 41.04) mm, rotated rx -180 ry 0 rz -180 deg; joints [-52.638, -9.48, 76.969, 73.705, 55.902, -62.46]
  Call Extruder(391.72493)
  MoveL 2278 to (-29.38, 163.88, 41.04) mm, rotated rx 180 ry 0 rz 180 deg; joints [-52.659, -9.503, 76.987, 73.714, 55.922, -62.463]
  MoveL 2279 to (-29.38, 163.88, 41.04) mm, rotated rx 180 ry 0 rz 180 deg; joints [-52.659, -9.503, 76.987, 73.714, 55.922, -62.463]
  Call Extruder(391.84000)
  MoveL 2280 to (-29.59, 163.84, 41.04) mm, rotated rx -180 ry 0 rz 180 deg; joints [-52.681, -9.526, 77.006, 73.724, 55.943, -62.465]
  MoveL 2281 to (-29.59, 163.84, 41.04) mm, rotated rx -180 ry 0 rz 180 deg; joints [-52.681, -9.526, 77.006, 73.724, 55.943, -62.465]
  Call Extruder(391.96224)
  MoveL 2282 to (-29.8, 163.78, 41.04) mm, rotated rx -180 ry 0 rz 180 deg; joints [-52.703, -9.55, 77.026, 73.733, 55.964, -62.467]
  MoveL 2283 to (-29.8, 163.78, 41.04) mm, rotated rx -180 ry 0 rz 180 deg; joints [-52.703, -9.55, 77.026, 73.733, 55.964, -62.467]
  Call Extruder(392.09192)
  MoveL 2284 to (-30.02, 163.72, 41.04) mm, rotated rx 180 ry 0 rz 180 deg; joints [-52.726, -9.577, 77.049, 73.743, 55.985, -62.468]
  MoveL 2285 to (-30.02, 163.72, 41.04) mm, rotated rx 180 ry 0 rz 180 deg; joints [-52.726, -9.577, 77.049, 73.743, 55.985, -62.468]
  Call Extruder(392.22216)
  MoveL 2286 to (-30.25, 163.65, 41.04) mm, rotated rx 180 ry 0 rz -180 deg; joints [-52.748, -9.604, 77.071, 73.752, 56.006, -62.469]
  MoveL 2287 to (-30.25, 163.65, 41.04) mm, rotated rx 180 ry 0 rz -180 deg; joints [-52.748, -9.604, 77.071, 73.752, 56.006, -62.469]
  Call Extruder(392.35297)
  MoveL 2288 to (-30.47, 163.58, 41.04) mm, rotated rx 180 ry 0 rz -180 deg; joints [-52.77, -9.631, 77.093, 73.761, 56.027, -62.471]
  MoveL 2289 to (-30.47, 163.58, 41.04) mm, rotated rx 180 ry 0 rz -180 deg; joints [-52.77, -9.631, 77.093, 73.761, 56.027, -62.471]
  Call Extruder(392.48435)
  MoveL 2290 to (-30.7, 163.51, 41.04) mm, rotated rx 180 ry 0 rz -180 deg; joints [-52.792, -9.658, 77.115, 73.77, 56.048, -62.472]
  MoveL 2291 to (-30.7, 163.51, 41.04) mm, rotated rx 180 ry 0 rz -180 deg; joints [-52.792, -9.658, 77.115, 73.77, 56.048, -62.472]
  Call Extruder(392.59624)
  MoveL 2292 to (-30.88, 163.45, 41.04) mm, rotated rx -180 ry 0 rz -180 deg; joints [-52.81, -9.681, 77.134, 73.778, 56.065, -62.473]
  MoveL 2293 to (-30.88, 163.45, 41.04) mm, rotated rx -180 ry 0 rz -180 deg; joints [-52.81, -9.681, 77.134, 73.778, 56.065, -62.473]
  Call Extruder(392.70858)
  MoveL 2294 to (-31.07, 163.39, 41.04) mm, rotated rx 180 ry 0 rz 180 deg; joints [-52.829, -9.704, 77.153, 73.786, 56.083, -62.474]
  MoveL 2295 to (-31.07, 163.39, 41.04) mm, rotated rx 180 ry 0 rz 180 deg; joints [-52.829, -9.704, 77.153, 73.786, 56.083, -62.474]
  Call Extruder(392.82136)
  MoveL 2296 to (-31.26, 163.33, 41.03) mm, rotated rx 180 ry 0 rz 180 deg; joints [-52.847, -9.728, 77.172, 73.793, 56.1, -62.474]
  MoveL 2297 to (-31.26, 163.33, 41.03) mm, rotated rx 180 ry 0 rz 180 deg; joints [-52.847, -9.728, 77.172, 73.793, 56.1, -62.474]
  Call Extruder(392.93458)
  MoveL 2298 to (-31.45, 163.27, 41.04) mm, rotated rx 180 ry 0 rz 180 deg; joints [-52.866, -9.751, 77.191, 73.801, 56.118, -62.475]
  MoveL 2299 to (-31.45, 163.27, 41.04) mm, rotated rx 180 ry 0 rz 180 deg; joints [-52.866, -9.751, 77.191, 73.801, 56.118, -62.475]
  Call Extruder(393.04826)
  MoveL 2300 to (-31.64, 163.21, 41.04) mm, rotated rx -180 ry 0 rz 180 deg; joints [-52.884, -9.774, 77.209, 73.808, 56.135, -62.476]
  MoveL 2301 to (-31.64, 163.21, 41.04) mm, rotated rx -180 ry 0 rz 180 deg; joints [-52.884, -9.774, 77.209, 73.808, 56.135, -62.476]
  Call Extruder(393.23023)
  MoveL 2302 to (-31.93, 163.09, 41.04) mm, rotated rx -180 ry 0 rz 180 deg; joints [-52.91, -9.813, 77.241, 73.818, 56.16, -62.476]
  MoveL 2303 to (-31.93, 163.09, 41.04) mm, rotated rx -180 ry 0 rz 180 deg; joints [-52.91, -9.813, 77.241, 73.818, 56.16, -62.476]
  Call Extruder(393.41296)
  MoveL 2304 to (-32.22, 162.97, 41.04) mm, rotated rx 180 ry 0 rz -180 deg; joints [-52.936, -9.851, 77.273, 73.828, 56.185, -62.476]
  MoveL 2305 to (-32.22, 162.97, 41.04) mm, rotated rx 180 ry 0 rz -180 deg; joints [-52.936, -9.851, 77.273, 73.828, 56.185, -62.476]
  Call Extruder(393.58337)
  MoveL 2306 to (-32.49, 162.85, 41.04) mm, rotated rx 180 ry 0 rz 180 deg; joints [-52.96, -9.887, 77.302, 73.837, 56.208, -62.476]
  MoveL 2307 to (-32.49, 162.85, 41.04) mm, rotated rx 180 ry 0 rz 180 deg; joints [-52.96, -9.887, 77.302, 73.837, 56.208, -62.476]
  Call Extruder(393.74134)
  MoveL 2308 to (-32.74, 162.74, 41.03) mm, rotated rx -180 ry 0 rz 180 deg; joints [-52.982, -9.921, 77.329, 73.845, 56.229, -62.475]
  MoveL 2309 to (-32.74, 162.74, 41.03) mm, rotated rx -180 ry 0 rz 180 deg; joints [-52.982, -9.921, 77.329, 73.845, 56.229, -62.475]
  Call Extruder(393.89990)
  MoveL 2310 to (-32.99, 162.64, 41.04) mm, rotated rx -180 ry 0 rz -180 deg; joints [-53.004, -9.954, 77.356, 73.853, 56.251, -62.475]
  MoveL 2311 to (-32.99, 162.64, 41.04) mm, rotated rx -180 ry 0 rz -180 deg; joints [-53.004, -9.954, 77.356, 73.853, 56.251, -62.475]
  Call Extruder(394.10607)
  MoveL 2312 to (-33.29, 162.46, 41.04) mm, rotated rx 180 ry 0 rz 180 deg; joints [-53.026, -10, 77.394, 73.86, 56.273, -62.472]
  MoveL 2313 to (-33.29, 162.46, 41.04) mm, rotated rx 180 ry 0 rz 180 deg; joints [-53.026, -10, 77.394, 73.86, 56.273, -62.472]
  Call Extruder(394.31302)
  MoveL 2314 to (-33.6, 162.29, 41.04) mm, rotated rx 180 ry 0 rz 180 deg; joints [-53.049, -10.046, 77.431, 73.867, 56.295, -62.469]
  MoveL 2315 to (-33.6, 162.29, 41.04) mm, rotated rx 180 ry 0 rz 180 deg; joints [-53.049, -10.046, 77.431, 73.867, 56.295, -62.469]
  Call Extruder(394.52075)
  MoveL 2316 to (-33.9, 162.11, 41.04) mm, rotated rx -180 ry 0 rz 180 deg; joints [-53.071, -10.091, 77.468, 73.874, 56.318, -62.466]
  MoveL 2317 to (-33.9, 162.11, 41.04) mm, rotated rx -180 ry 0 rz 180 deg; joints [-53.071, -10.091, 77.468, 73.874, 56.318, -62.466]
  Call Extruder(394.72926)
  MoveL 2318 to (-34.21, 161.94, 41.04) mm, rotated rx 180 ry 0 rz 180 deg; joints [-53.094, -10.137, 77.505, 73.881, 56.34, -62.463]
  MoveL 2319 to (-34.21, 161.94, 41.04) mm, rotated rx 180 ry 0 rz 180 deg; joints [-53.094, -10.137, 77.505, 73.881, 56.34, -62.463]
  Call Extruder(394.90880)
  MoveL 2320 to (-34.45, 161.76, 41.04) mm, rotated rx 180 ry 0 rz 180 deg; joints [-53.109, -10.178, 77.538, 73.885, 56.355, -62.458]
  MoveL 2321 to (-34.45, 161.76, 41.04) mm, rotated rx 180 ry 0 rz 180 deg; joints [-53.109, -10.178, 77.538, 73.885, 56.355, -62.458]
  Call Extruder(395.24224)
  MoveL 2322 to (-34.9, 161.43, 41.04) mm, rotated rx -180 ry 0 rz 180 deg; joints [-53.135, -10.253, 77.599, 73.89, 56.383, -62.45]
  MoveL 2323 to (-34.9, 161.43, 41.04) mm, rotated rx -180 ry 0 rz 180 deg; joints [-53.135, -10.253, 77.599, 73.89, 56.383, -62.45]
  Call Extruder(395.57686)
  MoveL 2324 to (-35.35, 161.1, 41.04) mm, rotated rx -180 ry 0 rz -180 deg; joints [-53.163, -10.329, 77.66, 73.896, 56.411, -62.442]
  Call Extruder(396.40476)
  MoveL 2325 to (-36.39, 160.19, 41.04) mm, rotated rx 180 ry 0 rz 180 deg; joints [-53.209, -10.52, 77.814, 73.898, 56.463, -62.413]
  Call Extruder(397.03477)
  MoveL 2326 to (-37.09, 159.41, 41.04) mm, rotated rx 180 ry 0 rz 180 deg; joints [-53.224, -10.668, 77.932, 73.888, 56.484, -62.384]
  Call Extruder(397.38246)
  MoveL 2327 to (-37.45, 158.95, 41.04) mm, rotated rx 180 ry 0 rz 180 deg; joints [-53.227, -10.749, 77.998, 73.879, 56.491, -62.366]
  MoveL 2328 to (-37.45, 158.95, 41.04) mm, rotated rx 180 ry 0 rz 180 deg; joints [-53.227, -10.749, 77.998, 73.879, 56.491, -62.366]
  Call Extruder(397.68150)
  MoveL 2329 to (-37.74, 158.55, 41.04) mm, rotated rx -180 ry 0 rz 180 deg; joints [-53.226, -10.82, 78.054, 73.869, 56.494, -62.349]
  MoveL 2330 to (-37.74, 158.55, 41.04) mm, rotated rx -180 ry 0 rz 180 deg; joints [-53.226, -10.82, 78.054, 73.869, 56.494, -62.349]
  Call Extruder(397.80380)
  MoveL 2331 to (-37.87, 158.38, 41.04) mm, rotated rx 180 ry 0 rz 180 deg; joints [-53.225, -10.849, 78.077, 73.865, 56.495, -62.342]
  Set speed (130.0 mm/s)
  MoveL 2332 to (-39.5, 155.47, 41.04) mm, rotated rx 180 ry 0 rz 180 deg; joints [-53.153, -11.313, 78.445, 73.764, 56.458, -62.209]
  Call M_RunCode(106)
  MoveL 2333 to (-39.5, 155.47, 50.44) mm, rotated rx 180 ry 0 rz 180 deg; joints [-53.153, -12.226, 80.739, 74.651, 56.082, -63.807]
  MoveL 2334 to (-38.84, 156.79, 50.44) mm, rotated rx -180 ry 0 rz 180 deg; joints [-53.196, -12.022, 80.581, 74.703, 56.109, -63.872]
  Set speed (30.0 mm/s)
  MoveL 2335 to (-38.84, 156.79, 50.44) mm, rotated rx -180 ry 0 rz 180 deg; joints [-53.196, -12.022, 80.581, 74.703, 56.109, -63.872]
  Call Extruder(397.96209)
  MoveL 2336 to (-38.94, 156.54, 50.44) mm, rotated rx 180 ry 0 rz 180 deg; joints [-53.186, -12.059, 80.609, 74.692, 56.102, -63.86]
  MoveL 2337 to (-38.94, 156.54, 50.44) mm, rotated rx 180 ry 0 rz 180 deg; joints [-53.186, -12.059, 80.609, 74.692, 56.102, -63.86]
  Call Extruder(398.11977)
  MoveL 2338 to (-39.05, 156.29, 50.44) mm, rotated rx 180 ry 0 rz 180 deg; joints [-53.175, -12.096, 80.638, 74.681, 56.094, -63.847]
  MoveL 2339 to (-39.05, 156.29, 50.44) mm, rotated rx 180 ry 0 rz 180 deg; joints [-53.175, -12.096, 80.638, 74.681, 56.094, -63.847]
  Call Extruder(398.28986)
  MoveL 2340 to (-39.16, 156.02, 50.44) mm, rotated rx 180 ry 0 rz 180 deg; joints [-53.163, -12.136, 80.669, 74.669, 56.086, -63.833]
  MoveL 2341 to (-39.16, 156.02, 50.44) mm, rotated rx 180 ry 0 rz 180 deg; joints [-53.163, -12.136, 80.669, 74.669, 56.086, -63.833]
  Call Extruder(398.47220)
  MoveL 2342 to (-39.29, 155.73, 50.44) mm, rotated rx 180 ry 0 rz 180 deg; joints [-53.15, -12.179, 80.703, 74.656, 56.077, -63.818]
  MoveL 2343 to (-39.29, 155.73, 50.44) mm, rotated rx 180 ry 0 rz 180 deg; joints [-53.15, -12.179, 80.703, 74.656, 56.077, -63.818]
  Call Extruder(398.65378)
  MoveL 2344 to (-39.41, 155.44, 50.44) mm, rotated rx -180 ry 0 rz 180 deg; joints [-53.137, -12.222, 80.736, 74.643, 56.068, -63.803]
  MoveL 2345 to (-39.41, 155.44, 50.44) mm, rotated rx -180 ry 0 rz 180 deg; joints [-53.137, -12.222, 80.736, 74.643, 56.068, -63.803]
  Call Extruder(398.76724)
  MoveL 2346 to (-39.47, 155.25, 50.44) mm, rotated rx 180 ry 0 rz -180 deg; joints [-53.126, -12.248, 80.756, 74.633, 56.059, -63.793]
  MoveL 2347 to (-39.47, 155.25, 50.44) mm, rotated rx 180 ry 0 rz -180 deg; joints [-53.126, -12.248, 80.756, 74.633, 56.059, -63.793]
  Call Extruder(398.88025)
  MoveL 2348 to (-39.53, 155.06, 50.44) mm, rotated rx -180 ry 0 rz -180 deg; joints [-53.115, -12.275, 80.777, 74.624, 56.051, -63.783]
  MoveL 2349 to (-39.53, 155.06, 50.44) mm, rotated rx -180 ry 0 rz -180 deg; joints [-53.115, -12.275, 80.777, 74.624, 56.051, -63.783]
  Call Extruder(398.99282)
  MoveL 2350 to (-39.59, 154.87, 50.44) mm, rotated rx 180 ry 0 rz 180 deg; joints [-53.105, -12.301, 80.797, 74.614, 56.043, -63.773]
  MoveL 2351 to (-39.59, 154.87, 50.44) mm, rotated rx 180 ry 0 rz 180 deg; joints [-53.105, -12.301, 80.797, 74.614, 56.043, -63.773]
  Call Extruder(399.10494)
  MoveL 2352 to (-39.65, 154.68, 50.44) mm, rotated rx -180 ry 0 rz 180 deg; joints [-53.094, -12.327, 80.817, 74.605, 56.035, -63.763]
  MoveL 2353 to (-39.65, 154.68, 50.44) mm, rotated rx -180 ry 0 rz 180 deg; joints [-53.094, -12.327, 80.817, 74.605, 56.035, -63.763]
  Call Extruder(399.21662)
  MoveL 2354 to (-39.71, 154.49, 50.44) mm, rotated rx 180 ry 0 rz 180 deg; joints [-53.083, -12.353, 80.837, 74.595, 56.027, -63.752]
  MoveL 2355 to (-39.71, 154.49, 50.44) mm, rotated rx 180 ry 0 rz 180 deg; joints [-53.083, -12.353, 80.837, 74.595, 56.027, -63.752]
  Call Extruder(399.34770)
  MoveL 2356 to (-39.78, 154.27, 50.44) mm, rotated rx 180 ry 0 rz 180 deg; joints [-53.069, -12.384, 80.861, 74.583, 56.017, -63.74]
  MoveL 2357 to (-39.78, 154.27, 50.44) mm, rotated rx 180 ry 0 rz 180 deg; joints [-53.069, -12.384, 80.861, 74.583, 56.017, -63.74]
  Call Extruder(399.47821)
  MoveL 2358 to (-39.85, 154.05, 50.44) mm, rotated rx -180 ry 0 rz -180 deg; joints [-53.056, -12.415, 80.885, 74.571, 56.006, -63.728]
  MoveL 2359 to (-39.85, 154.05, 50.44) mm, rotated rx -180 ry 0 rz -180 deg; joints [-53.056, -12.415, 80.885, 74.571, 56.006, -63.728]
  Call Extruder(399.60815)
  MoveL 2360 to (-39.92, 153.82, 50.44) mm, rotated rx 180 ry 0 rz -180 deg; joints [-53.042, -12.445, 80.909, 74.56, 55.996, -63.716]
  MoveL 2361 to (-39.92, 153.82, 50.44) mm, rotated rx 180 ry 0 rz -180 deg; joints [-53.042, -12.445, 80.909, 74.56, 55.996, -63.716]
  Call Extruder(399.73753)
  MoveL 2362 to (-39.98, 153.6, 50.44) mm, rotated rx 180 ry 0 rz 180 deg; joints [-53.029, -12.476, 80.932, 74.548, 55.986, -63.704]
  MoveL 2363 to (-39.98, 153.6, 50.44) mm, rotated rx 180 ry 0 rz 180 deg; joints [-53.029, -12.476, 80.932, 74.548, 55.986, -63.704]
  Call Extruder(399.85951)
  MoveL 2364 to (-40.04, 153.39, 50.44) mm, rotated rx 180 ry 0 rz -180 deg; joints [-53.015, -12.505, 80.954, 74.536, 55.975, -63.692]
  MoveL 2365 to (-40.04, 153.39, 50.44) mm, rotated rx 180 ry 0 rz -180 deg; joints [-53.015, -12.505, 80.954, 74.536, 55.975, -63.692]
  Call Extruder(399.97437)
  MoveL 2366 to (-40.08, 153.18, 50.44) mm, rotated rx 180 ry 0 rz -180 deg; joints [-53, -12.531, 80.975, 74.524, 55.963, -63.68]
  MoveL 2367 to (-40.08, 153.18, 50.44) mm, rotated rx 180 ry 0 rz -180 deg; joints [-53, -12.531, 80.975, 74.524, 55.963, -63.68]
  Call Extruder(400.08877)
  MoveL 2368 to (-40.13, 152.98, 50.44) mm, rotated rx 180 ry 0 rz 180 deg; joints [-52.985, -12.558, 80.995, 74.512, 55.952, -63.669]
  MoveL 2369 to (-40.13, 152.98, 50.44) mm, rotated rx 180 ry 0 rz 180 deg; joints [-52.985, -12.558, 80.995, 74.512, 55.952, -63.669]
  Call Extruder(400.20273)
  MoveL 2370 to (-40.17, 152.77, 50.44) mm, rotated rx -180 ry 0 rz 180 deg; joints [-52.97, -12.585, 81.016, 74.5, 55.94, -63.657]
  MoveL 2371 to (-40.17, 152.77, 50.44) mm, rotated rx -180 ry 0 rz 180 deg; joints [-52.97, -12.585, 81.016, 74.5, 55.94, -63.657]
  Call Extruder(400.31623)
  MoveL 2372 to (-40.22, 152.57, 50.44) mm, rotated rx 180 ry 0 rz 180 deg; joints [-52.956, -12.611, 81.036, 74.488, 55.929, -63.646]
  MoveL 2373 to (-40.22, 152.57, 50.44) mm, rotated rx 180 ry 0 rz 180 deg; joints [-52.956, -12.611, 81.036, 74.488, 55.929, -63.646]
  Call Extruder(400.45351)
  MoveL 2374 to (-40.27, 152.32, 50.44) mm, rotated rx 180 ry 0 rz 180 deg; joints [-52.937, -12.643, 81.06, 74.474, 55.914, -63.631]
  MoveL 2375 to (-40.27, 152.32, 50.44) mm, rotated rx 180 ry 0 rz 180 deg; joints [-52.937, -12.643, 81.06, 74.474, 55.914, -63.631]
  Call Extruder(400.59019)
  MoveL 2376 to (-40.32, 152.07, 50.44) mm, rotated rx -180 ry 0 rz -180 deg; joints [-52.918, -12.675, 81.085, 74.459, 55.899, -63.617]
  MoveL 2377 to (-40.32, 152.07, 50.44) mm, rotated rx -180 ry 0 rz -180 deg; joints [-52.918, -12.675, 81.085, 74.459, 55.899, -63.617]
  Call Extruder(400.72625)
  MoveL 2378 to (-40.37, 151.82, 50.44) mm, rotated rx 180 ry 0 rz 180 deg; joints [-52.9, -12.707, 81.109, 74.444, 55.884, -63.603]
  MoveL 2379 to (-40.37, 151.82, 50.44) mm, rotated rx 180 ry 0 rz 180 deg; joints [-52.9, -12.707, 81.109, 74.444, 55.884, -63.603]
  Call Extruder(400.86170)
  MoveL 2380 to (-40.42, 151.57, 50.44) mm, rotated rx 180 ry 0 rz 180 deg; joints [-52.881, -12.739, 81.134, 74.429, 55.869, -63.588]
  MoveL 2381 to (-40.42, 151.57, 50.44) mm, rotated rx 180 ry 0 rz 180 deg; joints [-52.881, -12.739, 81.134, 74.429, 55.869, -63.588]
  Call Extruder(400.99654)
  MoveL 2382 to (-40.47, 151.32, 50.44) mm, rotated rx 180 ry 0 rz 180 deg; joints [-52.862, -12.77, 81.158, 74.414, 55.855, -63.574]
  MoveL 2383 to (-40.47, 151.32, 50.44) mm, rotated rx 180 ry 0 rz 180 deg; joints [-52.862, -12.77, 81.158, 74.414, 55.855, -63.574]
  Call Extruder(401.13077)
  MoveL 2384 to (-40.52, 151.08, 50.44) mm, rotated rx 180 ry 0 rz 180 deg; joints [-52.843, -12.802, 81.183, 74.399, 55.84, -63.56]
  MoveL 2385 to (-40.52, 151.08, 50.44) mm, rotated rx 180 ry 0 rz 180 deg; joints [-52.843, -12.802, 81.183, 74.399, 55.84, -63.56]
  Call Extruder(401.26438)
  MoveL 2386 to (-40.56, 150.83, 50.44) mm, rotated rx 180 ry 0 rz 180 deg; joints [-52.824, -12.834, 81.207, 74.384, 55.825, -63.545]
  MoveL 2387 to (-40.56, 150.83, 50.44) mm, rotated rx 180 ry 0 rz 180 deg; joints [-52.824, -12.834, 81.207, 74.384, 55.825, -63.545]
  Call Extruder(401.42647)
  MoveL 2388 to (-40.61, 150.52, 50.44) mm, rotated rx 180 ry 0 rz 180 deg; joints [-52.799, -12.872, 81.236, 74.364, 55.805, -63.527]
  MoveL 2389 to (-40.61, 150.52, 50.44) mm, rotated rx 180 ry 0 rz 180 deg; joints [-52.799, -12.872, 81.236, 74.364, 55.805, -63.527]
  Call Extruder(401.58783)
  MoveL 2390 to (-40.66, 150.21, 50.44) mm, rotated rx 180 ry 0 rz -180 deg; joints [-52.775, -12.91, 81.265, 74.345, 55.785, -63.509]
  MoveL 2391 to (-40.66, 150.21, 50.44) mm, rotated rx 180 ry 0 rz -180 deg; joints [-52.775, -12.91, 81.265, 74.345, 55.785, -63.509]
  Call Extruder(401.74847)
  MoveL 2392 to (-40.71, 149.91, 50.44) mm, rotated rx 180 ry 0 rz 180 deg; joints [-52.75, -12.948, 81.294, 74.326, 55.766, -63.491]
  MoveL 2393 to (-40.71, 149.91, 50.44) mm, rotated rx 180 ry 0 rz 180 deg; joints [-52.75, -12.948, 81.294, 74.326, 55.766, -63.491]
  Call Extruder(401.90837)
  MoveL 2394 to (-40.76, 149.6, 50.44) mm, rotated rx 180 ry 0 rz 180 deg; joints [-52.725, -12.986, 81.323, 74.306, 55.746, -63.473]
  MoveL 2395 to (-40.76, 149.6, 50.44) mm, rotated rx 180 ry 0 rz 180 deg; joints [-52.725, -12.986, 81.323, 74.306, 55.746, -63.473]
  Call Extruder(402.06755)
  MoveL 2396 to (-40.81, 149.3, 50.44) mm, rotated rx 180 ry 0 rz 180 deg; joints [-52.7, -13.024, 81.352, 74.287, 55.726, -63.455]
  MoveL 2397 to (-40.81, 149.3, 50.44) mm, rotated rx 180 ry 0 rz 180 deg; joints [-52.7, -13.024, 81.352, 74.287, 55.726, -63.455]
  Call Extruder(402.22600)
  MoveL 2398 to (-40.86, 148.99, 50.44) mm, rotated rx -180 ry 0 rz -180 deg; joints [-52.675, -13.062, 81.381, 74.267, 55.706, -63.436]
  MoveL 2399 to (-40.86, 148.99, 50.44) mm, rotated rx -180 ry 0 rz -180 deg; joints [-52.675, -13.062, 81.381, 74.267, 55.706, -63.436]
  Call Extruder(402.42488)
  MoveL 2400 to (-40.9, 148.6, 50.44) mm, rotated rx 180 ry 0 rz 180 deg; joints [-52.641, -13.109, 81.416, 74.242, 55.679, -63.413]
  MoveL 2401 to (-40.9, 148.6, 50.44) mm, rotated rx 180 ry 0 rz 180 deg; joints [-52.641, -13.109, 81.416, 74.242, 55.679, -63.413]
  Call Extruder(402.62289)
  MoveL 2402 to (-40.95, 148.22, 50.44) mm, rotated rx 180 ry 0 rz 180 deg; joints [-52.607, -13.156, 81.452, 74.216, 55.651, -63.389]
  MoveL 2403 to (-40.95, 148.22, 50.44) mm, rotated rx 180 ry 0 rz 180 deg; joints [-52.607, -13.156, 81.452, 74.216, 55.651, -63.389]
  Call Extruder(402.82003)
  MoveL 2404 to (-40.99, 147.83, 50.44) mm, rotated rx 180 ry 0 rz 180 deg; joints [-52.573, -13.202, 81.487, 74.19, 55.624, -63.366]
  MoveL 2405 to (-40.99, 147.83, 50.44) mm, rotated rx 180 ry 0 rz 180 deg; joints [-52.573, -13.202, 81.487, 74.19, 55.624, -63.366]
  Call Extruder(403.01630)
  MoveL 2406 to (-41.04, 147.44, 50.44) mm, rotated rx 180 ry 0 rz 180 deg; joints [-52.539, -13.249, 81.522, 74.164, 55.596, -63.342]
  MoveL 2407 to (-41.04, 147.44, 50.44) mm, rotated rx 180 ry 0 rz 180 deg; joints [-52.539, -13.249, 81.522, 74.164, 55.596, -63.342]
  Call Extruder(403.26199)
  MoveL 2408 to (-41.09, 146.95, 50.44) mm, rotated rx 180 ry 0 rz 180 deg; joints [-52.494, -13.307, 81.566, 74.13, 55.56, -63.312]
  MoveL 2409 to (-41.09, 146.95, 50.44) mm, rotated rx 180 ry 0 rz 180 deg; joints [-52.494, -13.307, 81.566, 74.13, 55.56, -63.312]
  Call Extruder(403.55672)
  MoveL 2410 to (-41.13, 146.36, 50.44) mm, rotated rx 180 ry 0 rz 180 deg; joints [-52.439, -13.375, 81.618, 74.089, 55.516, -63.275]
  MoveL 2411 to (-41.13, 146.36, 50.44) mm, rotated rx 180 ry 0 rz 180 deg; joints [-52.439, -13.375, 81.618, 74.089, 55.516, -63.275]
  Call Extruder(403.85012)
  MoveL 2412 to (-41.18, 145.77, 50.44) mm, rotated rx 180 ry 0 rz 180 deg; joints [-52.383, -13.444, 81.669, 74.047, 55.471, -63.238]
  MoveL 2413 to (-41.18, 145.77, 50.44) mm, rotated rx 180 ry 0 rz 180 deg; joints [-52.383, -13.444, 81.669, 74.047, 55.471, -63.238]
  Call Extruder(404.28345)
  MoveL 2414 to (-41.22, 144.9, 50.44) mm, rotated rx 180 ry 0 rz -180 deg; joints [-52.297, -13.544, 81.745, 73.984, 55.401, -63.182]
  MoveL 2415 to (-41.22, 144.9, 50.44) mm, rotated rx 180 ry 0 rz -180 deg; joints [-52.297, -13.544, 81.745, 73.984, 55.401, -63.182]
  Call Extruder(404.85561)
  MoveL 2416 to (-41.27, 143.74, 50.44) mm, rotated rx 180 ry 0 rz -180 deg; joints [-52.18, -13.676, 81.843, 73.898, 55.306, -63.107]
  MoveL 2417 to (-41.27, 143.74, 50.44) mm, rotated rx 180 ry 0 rz -180 deg; joints [-52.18, -13.676, 81.843, 73.898, 55.306, -63.107]
  Call Extruder(405.28344)
  MoveL 2418 to (-41.29, 142.86, 50.44) mm, rotated rx 180 ry 0 rz 180 deg; joints [-52.09, -13.773, 81.915, 73.832, 55.232, -63.05]
  Call Extruder(447.27697)
  MoveL 2419 to (-41.29, 57.14, 50.44) mm, rotated rx 180 ry 0 rz 180 deg; joints [-40.759, -22.129, 87.481, 64.18, 46.492, -54.9]
  MoveL 2420 to (-41.29, 57.14, 50.44) mm, rotated rx 180 ry 0 rz 180 deg; joints [-40.759, -22.129, 87.481, 64.18, 46.492, -54.9]
  Call Extruder(447.99254)
  MoveL 2421 to (-41.25, 55.68, 50.44) mm, rotated rx -180 ry 0 rz 180 deg; joints [-40.517, -22.247, 87.55, 63.945, 46.316, -54.706]
  MoveL 2422 to (-41.25, 55.68, 50.44) mm, rotated rx -180 ry 0 rz 180 deg; joints [-40.517, -22.247, 87.55, 63.945, 46.316, -54.706]
  Call Extruder(448.56728)
  MoveL 2423 to (-41.2, 54.52, 50.44) mm, rotated rx 180 ry 0 rz 180 deg; joints [-40.32, -22.34, 87.604, 63.754, 46.173, -54.549]
  MoveL 2424 to (-41.2, 54.52, 50.44) mm, rotated rx 180 ry 0 rz 180 deg; joints [-40.32, -22.34, 87.604, 63.754, 46.173, -54.549]
  Call Extruder(448.86068)
  MoveL 2425 to (-41.15, 53.93, 50.44) mm, rotated rx 180 ry 0 rz 180 deg; joints [-40.217, -22.385, 87.63, 63.655, 46.097, -54.468]
  MoveL 2426 to (-41.15, 53.93, 50.44) mm, rotated rx 180 ry 0 rz 180 deg; joints [-40.217, -22.385, 87.63, 63.655, 46.097, -54.468]
  Call Extruder(449.15541)
  MoveL 2427 to (-41.11, 53.34, 50.44) mm, rotated rx 180 ry 0 rz 180 deg; joints [-40.114, -22.429, 87.656, 63.555, 46.022, -54.386]
  MoveL 2428 to (-41.11, 53.34, 50.44) mm, rotated rx 180 ry 0 rz 180 deg; joints [-40.114, -22.429, 87.656, 63.555, 46.022, -54.386]
  Call Extruder(449.45147)
  MoveL 2429 to (-41.06, 52.75, 50.44) mm, rotated rx 180 ry 0 rz 180 deg; joints [-40.01, -22.474, 87.681, 63.455, 45.946, -54.304]
  MoveL 2430 to (-41.06, 52.75, 50.44) mm, rotated rx 180 ry 0 rz 180 deg; joints [-40.01, -22.474, 87.681, 63.455, 45.946, -54.304]
  Call Extruder(449.64774)
  MoveL 2431 to (-41.02, 52.37, 50.44) mm, rotated rx 180 ry 0 rz 180 deg; joints [-39.939, -22.502, 87.697, 63.387, 45.894, -54.25]
  MoveL 2432 to (-41.02, 52.37, 50.44) mm, rotated rx 180 ry 0 rz 180 deg; joints [-39.939, -22.502, 87.697, 63.387, 45.894, -54.25]
  Call Extruder(449.84488)
  MoveL 2433 to (-40.97, 51.98, 50.44) mm, rotated rx 180 ry 0 rz 180 deg; joints [-39.869, -22.529, 87.713, 63.32, 45.842, -54.195]
  MoveL 2434 to (-40.97, 51.98, 50.44) mm, rotated rx 180 ry 0 rz 180 deg; joints [-39.869, -22.529, 87.713, 63.32, 45.842, -54.195]
  Call Extruder(450.04289)
  MoveL 2435 to (-40.93, 51.59, 50.44) mm, rotated rx 180 ry 0 rz 180 deg; joints [-39.798, -22.557, 87.729, 63.252, 45.79, -54.141]
  MoveL 2436 to (-40.93, 51.59, 50.44) mm, rotated rx 180 ry 0 rz 180 deg; joints [-39.798, -22.557, 87.729, 63.252, 45.79, -54.141]
  Call Extruder(450.24176)
  MoveL 2437 to (-40.88, 51.2, 50.44) mm, rotated rx 180 ry 0 rz 180 deg; joints [-39.727, -22.584, 87.745, 63.184, 45.737, -54.086]
  MoveL 2438 to (-40.88, 51.2, 50.44) mm, rotated rx 180 ry 0 rz 180 deg; joints [-39.727, -22.584, 87.745, 63.184, 45.737, -54.086]
  Call Extruder(450.42084)
  MoveL 2439 to (-40.83, 50.86, 50.44) mm, rotated rx 180 ry 0 rz 180 deg; joints [-39.663, -22.608, 87.758, 63.122, 45.69, -54.036]
  MoveL 2440 to (-40.83, 50.86, 50.44) mm, rotated rx 180 ry 0 rz 180 deg; joints [-39.663, -22.608, 87.758, 63.122, 45.69, -54.036]
  Call Extruder(450.58002)
  MoveL 2441 to (-40.78, 50.55, 50.44) mm, rotated rx 180 ry 0 rz 180 deg; joints [-39.605, -22.628, 87.77, 63.067, 45.647, -53.992]
  MoveL 2442 to (-40.78, 50.55, 50.44) mm, rotated rx 180 ry 0 rz 180 deg; joints [-39.605, -22.628, 87.77, 63.067, 45.647, -53.992]
  Call Extruder(450.73993)
  MoveL 2443 to (-40.74, 50.24, 50.44) mm, rotated rx -180 ry 0 rz 180 deg; joints [-39.547, -22.649, 87.782, 63.012, 45.604, -53.948]
  MoveL 2444 to (-40.74, 50.24, 50.44) mm, rotated rx -180 ry 0 rz 180 deg; joints [-39.547, -22.649, 87.782, 63.012, 45.604, -53.948]
  Call Extruder(450.90057)
  MoveL 2445 to (-40.69, 49.94, 50.44) mm, rotated rx -180 ry 0 rz 180 deg; joints [-39.489, -22.669, 87.793, 62.957, 45.561, -53.904]
  MoveL 2446 to (-40.69, 49.94, 50.44) mm, rotated rx -180 ry 0 rz 180 deg; joints [-39.489, -22.669, 87.793, 62.957, 45.561, -53.904]
  Call Extruder(451.06193)
  MoveL 2447 to (-40.64, 49.63, 50.44) mm, rotated rx 180 ry 0 rz 180 deg; joints [-39.431, -22.689, 87.805, 62.901, 45.519, -53.86]
  MoveL 2448 to (-40.64, 49.63, 50.44) mm, rotated rx 180 ry 0 rz 180 deg; joints [-39.431, -22.689, 87.805, 62.901, 45.519, -53.86]
  Call Extruder(451.22402)
  MoveL 2449 to (-40.59, 49.33, 50.44) mm, rotated rx 180 ry 0 rz 180 deg; joints [-39.373, -22.709, 87.817, 62.846, 45.476, -53.815]
  MoveL 2450 to (-40.59, 49.33, 50.44) mm, rotated rx 180 ry 0 rz 180 deg; joints [-39.373, -22.709, 87.817, 62.846, 45.476, -53.815]
  Call Extruder(451.37222)
  MoveL 2451 to (-40.54, 49.05, 50.44) mm, rotated rx 180 ry 0 rz 180 deg; joints [-39.32, -22.727, 87.827, 62.795, 45.436, -53.775]
  MoveL 2452 to (-40.54, 49.05, 50.44) mm, rotated rx 180 ry 0 rz 180 deg; joints [-39.32, -22.727, 87.827, 62.795, 45.436, -53.775]
  Call Extruder(451.50645)
  MoveL 2453 to (-40.49, 48.8, 50.44) mm, rotated rx 180 ry 0 rz -180 deg; joints [-39.271, -22.742, 87.836, 62.749, 45.4, -53.738]
  MoveL 2454 to (-40.49, 48.8, 50.44) mm, rotated rx 180 ry 0 rz -180 deg; joints [-39.271, -22.742, 87.836, 62.749, 45.4, -53.738]
  Call Extruder(451.64129)
  MoveL 2455 to (-40.44, 48.55, 50.44) mm, rotated rx 180 ry 0 rz 180 deg; joints [-39.222, -22.758, 87.844, 62.702, 45.363, -53.702]
  MoveL 2456 to (-40.44, 48.55, 50.44) mm, rotated rx 180 ry 0 rz 180 deg; joints [-39.222, -22.758, 87.844, 62.702, 45.363, -53.702]
  Call Extruder(451.77674)
  MoveL 2457 to (-40.39, 48.3, 50.44) mm, rotated rx 180 ry 0 rz 180 deg; joints [-39.174, -22.773, 87.853, 62.656, 45.327, -53.665]
  MoveL 2458 to (-40.39, 48.3, 50.44) mm, rotated rx 180 ry 0 rz 180 deg; joints [-39.174, -22.773, 87.853, 62.656, 45.327, -53.665]
  Call Extruder(451.91280)
  MoveL 2459 to (-40.34, 48.05, 50.44) mm, rotated rx -180 ry 0 rz -180 deg; joints [-39.125, -22.788, 87.862, 62.609, 45.291, -53.628]
  MoveL 2460 to (-40.34, 48.05, 50.44) mm, rotated rx -180 ry 0 rz -180 deg; joints [-39.125, -22.788, 87.862, 62.609, 45.291, -53.628]
  Call Extruder(452.04947)
  MoveL 2461 to (-40.29, 47.8, 50.44) mm, rotated rx 180 ry 0 rz 180 deg; joints [-39.076, -22.804, 87.871, 62.563, 45.254, -53.591]
  MoveL 2462 to (-40.29, 47.8, 50.44) mm, rotated rx 180 ry 0 rz 180 deg; joints [-39.076, -22.804, 87.871, 62.563, 45.254, -53.591]
  Call Extruder(452.18675)
  MoveL 2463 to (-40.24, 47.56, 50.44) mm, rotated rx 180 ry 0 rz 180 deg; joints [-39.027, -22.819, 87.879, 62.516, 45.218, -53.554]
  MoveL 2464 to (-40.24, 47.56, 50.44) mm, rotated rx 180 ry 0 rz 180 deg; joints [-39.027, -22.819, 87.879, 62.516, 45.218, -53.554]
  Call Extruder(452.31242)
  MoveL 2465 to (-40.2, 47.33, 50.44) mm, rotated rx 180 ry 0 rz -180 deg; joints [-38.982, -22.833, 87.887, 62.473, 45.185, -53.52]
  MoveL 2466 to (-40.2, 47.33, 50.44) mm, rotated rx 180 ry 0 rz -180 deg; joints [-38.982, -22.833, 87.887, 62.473, 45.185, -53.52]
  Call Extruder(452.42638)
  MoveL 2467 to (-40.15, 47.12, 50.44) mm, rotated rx -180 ry 0 rz 180 deg; joints [-38.941, -22.845, 87.894, 62.434, 45.154, -53.489]
  MoveL 2468 to (-40.15, 47.12, 50.44) mm, rotated rx -180 ry 0 rz 180 deg; joints [-38.941, -22.845, 87.894, 62.434, 45.154, -53.489]
  Call Extruder(452.54078)
  MoveL 2469 to (-40.11, 46.92, 50.44) mm, rotated rx 180 ry 0 rz 180 deg; joints [-38.9, -22.857, 87.901, 62.396, 45.124, -53.459]
  MoveL 2470 to (-40.11, 46.92, 50.44) mm, rotated rx 180 ry 0 rz 180 deg; joints [-38.9, -22.857, 87.901, 62.396, 45.124, -53.459]
  Call Extruder(452.65564)
  MoveL 2471 to (-40.06, 46.72, 50.44) mm, rotated rx 180 ry 0 rz 180 deg; joints [-38.859, -22.869, 87.908, 62.357, 45.093, -53.428]
  MoveL 2472 to (-40.06, 46.72, 50.44) mm, rotated rx 180 ry 0 rz 180 deg; joints [-38.859, -22.869, 87.908, 62.357, 45.093, -53.428]
  Call Extruder(452.77095)
  MoveL 2473 to (-40.02, 46.51, 50.44) mm, rotated rx 180 ry 0 rz -180 deg; joints [-38.819, -22.881, 87.914, 62.318, 45.063, -53.397]
  MoveL 2474 to (-40.02, 46.51, 50.44) mm, rotated rx 180 ry 0 rz -180 deg; joints [-38.819, -22.881, 87.914, 62.318, 45.063, -53.397]
  Call Extruder(452.90034)
  MoveL 2475 to (-39.95, 46.29, 50.44) mm, rotated rx 180 ry 0 rz 180 deg; joints [-38.771, -22.892, 87.921, 62.273, 45.027, -53.363]
  MoveL 2476 to (-39.95, 46.29, 50.44) mm, rotated rx 180 ry 0 rz 180 deg; joints [-38.771, -22.892, 87.921, 62.273, 45.027, -53.363]
  Call Extruder(453.03028)
  MoveL 2477 to (-39.88, 46.06, 50.44) mm, rotated rx 180 ry 0 rz 180 deg; joints [-38.724, -22.903, 87.927, 62.229, 44.991, -53.329]
  MoveL 2478 to (-39.88, 46.06, 50.44) mm, rotated rx 180 ry 0 rz 180 deg; joints [-38.724, -22.903, 87.927, 62.229, 44.991, -53.329]
  Call Extruder(453.16079)
  MoveL 2479 to (-39.81, 45.84, 50.44) mm, rotated rx -180 ry 0 rz 180 deg; joints [-38.677, -22.914, 87.934, 62.185, 44.956, -53.294]
  MoveL 2480 to (-39.81, 45.84, 50.44) mm, rotated rx -180 ry 0 rz 180 deg; joints [-38.677, -22.914, 87.934, 62.185, 44.956, -53.294]
  Call Extruder(453.29187)
  MoveL 2481 to (-39.75, 45.62, 50.44) mm, rotated rx 180 ry 0 rz 180 deg; joints [-38.629, -22.926, 87.94, 62.14, 44.92, -53.26]
  MoveL 2482 to (-39.75, 45.62, 50.44) mm, rotated rx 180 ry 0 rz 180 deg; joints [-38.629, -22.926, 87.94, 62.14, 44.92, -53.26]
  Call Extruder(453.41351)
  MoveL 2483 to (-39.68, 45.41, 50.44) mm, rotated rx -180 ry 0 rz 180 deg; joints [-38.585, -22.936, 87.946, 62.099, 44.887, -53.228]
  MoveL 2484 to (-39.68, 45.41, 50.44) mm, rotated rx -180 ry 0 rz 180 deg; joints [-38.585, -22.936, 87.946, 62.099, 44.887, -53.228]
  Call Extruder(453.52564)
  MoveL 2485 to (-39.62, 45.22, 50.44) mm, rotated rx 180 ry 0 rz 180 deg; joints [-38.544, -22.945, 87.951, 62.061, 44.856, -53.199]
  MoveL 2486 to (-39.62, 45.22, 50.44) mm, rotated rx 180 ry 0 rz 180 deg; joints [-38.544, -22.945, 87.951, 62.061, 44.856, -53.199]
  Call Extruder(453.63821)
  MoveL 2487 to (-39.56, 45.03, 50.44) mm, rotated rx -180 ry 0 rz 180 deg; joints [-38.504, -22.954, 87.956, 62.023, 44.825, -53.169]
  MoveL 2488 to (-39.56, 45.03, 50.44) mm, rotated rx -180 ry 0 rz 180 deg; joints [-38.504, -22.954, 87.956, 62.023, 44.825, -53.169]
  Call Extruder(453.75122)
  MoveL 2489 to (-39.5, 44.85, 50.44) mm, rotated rx 180 ry 0 rz 180 deg; joints [-38.463, -22.962, 87.961, 61.985, 44.795, -53.14]
  MoveL 2490 to (-39.5, 44.85, 50.44) mm, rotated rx 180 ry 0 rz 180 deg; joints [-38.463, -22.962, 87.961, 61.985, 44.795, -53.14]
  Call Extruder(453.86468)
  MoveL 2491 to (-39.44, 44.66, 50.44) mm, rotated rx 180 ry 0 rz 180 deg; joints [-38.422, -22.971, 87.966, 61.947, 44.764, -53.11]
  MoveL 2492 to (-39.44, 44.66, 50.44) mm, rotated rx 180 ry 0 rz 180 deg; joints [-38.422, -22.971, 87.966, 61.947, 44.764, -53.11]
  Call Extruder(454.01232)
  MoveL 2493 to (-39.35, 44.42, 50.44) mm, rotated rx 180 ry 0 rz 180 deg; joints [-38.369, -22.981, 87.972, 61.898, 44.723, -53.073]
  MoveL 2494 to (-39.35, 44.42, 50.44) mm, rotated rx 180 ry 0 rz 180 deg; joints [-38.369, -22.981, 87.972, 61.898, 44.723, -53.073]
  Call Extruder(454.19466)
  MoveL 2495 to (-39.23, 44.13, 50.44) mm, rotated rx 180 ry 0 rz 180 deg; joints [-38.302, -22.992, 87.978, 61.836, 44.672, -53.026]
  MoveL 2496 to (-39.23, 44.13, 50.44) mm, rotated rx 180 ry 0 rz 180 deg; joints [-38.302, -22.992, 87.978, 61.836, 44.672, -53.026]
  Call Extruder(454.37775)
  MoveL 2497 to (-39.11, 43.83, 50.44) mm, rotated rx 180 ry 0 rz 180 deg; joints [-38.236, -23.004, 87.984, 61.775, 44.621, -52.979]
  MoveL 2498 to (-39.11, 43.83, 50.44) mm, rotated rx 180 ry 0 rz 180 deg; joints [-38.236, -23.004, 87.984, 61.775, 44.621, -52.979]
  Call Extruder(454.53544)
  MoveL 2499 to (-39, 43.58, 50.44) mm, rotated rx 180 ry 0 rz 180 deg; joints [-38.178, -23.012, 87.989, 61.722, 44.577, -52.939]
  MoveL 2500 to (-39, 43.58, 50.44) mm, rotated rx 180 ry 0 rz 180 deg; joints [-38.178, -23.012, 87.989, 61.722, 44.577, -52.939]
  Call Extruder(454.69372)
  MoveL 2501 to (-38.89, 43.33, 50.44) mm, rotated rx 180 ry 0 rz 180 deg; joints [-38.121, -23.021, 87.994, 61.669, 44.533, -52.899]
  MoveL 2502 to (-38.89, 43.33, 50.44) mm, rotated rx 180 ry 0 rz 180 deg; joints [-38.121, -23.021, 87.994, 61.669, 44.533, -52.899]
  Call Extruder(454.87574)
  MoveL 2503 to (-38.75, 43.06, 50.44) mm, rotated rx -180 ry 0 rz 180 deg; joints [-38.054, -23.029, 87.999, 61.609, 44.481, -52.854]
  MoveL 2504 to (-38.75, 43.06, 50.44) mm, rotated rx -180 ry 0 rz 180 deg; joints [-38.054, -23.029, 87.999, 61.609, 44.481, -52.854]
  Call Extruder(455.08230)
  MoveL 2505 to (-38.57, 42.75, 50.44) mm, rotated rx 180 ry 0 rz 180 deg; joints [-37.977, -23.035, 88.002, 61.541, 44.422, -52.804]
  MoveL 2506 to (-38.57, 42.75, 50.44) mm, rotated rx 180 ry 0 rz 180 deg; joints [-37.977, -23.035, 88.002, 61.541, 44.422, -52.804]
  Call Extruder(455.28963)
  MoveL 2507 to (-38.4, 42.45, 50.44) mm, rotated rx 180 ry 0 rz -180 deg; joints [-37.901, -23.042, 88.006, 61.472, 44.362, -52.753]
  MoveL 2508 to (-38.4, 42.45, 50.44) mm, rotated rx 180 ry 0 rz -180 deg; joints [-37.901, -23.042, 88.006, 61.472, 44.362, -52.753]
  Call Extruder(455.49774)
  MoveL 2509 to (-38.22, 42.15, 50.44) mm, rotated rx 180 ry 0 rz 180 deg; joints [-37.825, -23.048, 88.009, 61.404, 44.303, -52.702]
  MoveL 2510 to (-38.22, 42.15, 50.44) mm, rotated rx 180 ry 0 rz 180 deg; joints [-37.825, -23.048, 88.009, 61.404, 44.303, -52.702]
  Call Extruder(455.61546)
  MoveL 2511 to (-38.12, 41.97, 50.44) mm, rotated rx 180 ry 0 rz 180 deg; joints [-37.782, -23.051, 88.011, 61.365, 44.269, -52.674]
  MoveL 2512 to (-38.12, 41.97, 50.44) mm, rotated rx 180 ry 0 rz 180 deg; joints [-37.782, -23.051, 88.011, 61.365, 44.269, -52.674]
  Call Extruder(455.94830)
  MoveL 2513 to (-37.79, 41.52, 50.44) mm, rotated rx 180 ry 0 rz 180 deg; joints [-37.659, -23.053, 88.012, 61.257, 44.172, -52.596]
  MoveL 2514 to (-37.79, 41.52, 50.44) mm, rotated rx 180 ry 0 rz 180 deg; joints [-37.659, -23.053, 88.012, 61.257, 44.172, -52.596]
  Call Extruder(456.28234)
  MoveL 2515 to (-37.47, 41.07, 50.44) mm, rotated rx 180 ry 0 rz 180 deg; joints [-37.537, -23.055, 88.013, 61.15, 44.075, -52.518]
  MoveL 2516 to (-37.47, 41.07, 50.44) mm, rotated rx 180 ry 0 rz 180 deg; joints [-37.537, -23.055, 88.013, 61.15, 44.075, -52.518]
  Call Extruder(456.44993)
  MoveL 2517 to (-37.3, 40.85, 50.44) mm, rotated rx 180 ry 0 rz 180 deg; joints [-37.475, -23.056, 88.014, 61.096, 44.027, -52.479]
  Call Extruder(457.27924)
  MoveL 2518 to (-36.39, 39.81, 50.44) mm, rotated rx 180 ry 0 rz 180 deg; joints [-37.173, -23.044, 88.007, 60.834, 43.785, -52.294]
  Call Extruder(457.91031)
  MoveL 2519 to (-35.6, 39.11, 50.44) mm, rotated rx -180 ry 0 rz 180 deg; joints [-36.947, -23.017, 87.992, 60.644, 43.6, -52.164]
  MoveL 2520 to (-35.6, 39.11, 50.44) mm, rotated rx -180 ry 0 rz 180 deg; joints [-36.947, -23.017, 87.992, 60.644, 43.6, -52.164]
  Call Extruder(458.10788)
  MoveL 2521 to (-35.35, 38.9, 50.44) mm, rotated rx -180 ry 0 rz 180 deg; joints [-36.876, -23.008, 87.987, 60.585, 43.543, -52.123]
  Call Extruder(458.44190)
  MoveL 2522 to (-34.9, 38.57, 50.44) mm, rotated rx 180 ry 0 rz -180 deg; joints [-36.759, -22.987, 87.975, 60.489, 43.446, -52.059]
  MoveL 2523 to (-34.9, 38.57, 50.44) mm, rotated rx 180 ry 0 rz -180 deg; joints [-36.759, -22.987, 87.975, 60.489, 43.446, -52.059]
  Call Extruder(458.77473)
  MoveL 2524 to (-34.45, 38.24, 50.44) mm, rotated rx 180 ry 0 rz 180 deg; joints [-36.642, -22.965, 87.963, 60.393, 43.349, -51.995]
  MoveL 2525 to (-34.45, 38.24, 50.44) mm, rotated rx 180 ry 0 rz 180 deg; joints [-36.642, -22.965, 87.963, 60.393, 43.349, -51.995]
  Call Extruder(458.95398)
  MoveL 2526 to (-34.21, 38.07, 50.44) mm, rotated rx -180 ry 0 rz 180 deg; joints [-36.579, -22.954, 87.956, 60.341, 43.297, -51.96]
  MoveL 2527 to (-34.21, 38.07, 50.44) mm, rotated rx -180 ry 0 rz 180 deg; joints [-36.579, -22.954, 87.956, 60.341, 43.297, -51.96]
  Call Extruder(459.16208)
  MoveL 2528 to (-33.9, 37.89, 50.44) mm, rotated rx 180 ry 0 rz 180 deg; joints [-36.509, -22.936, 87.946, 60.285, 43.238, -51.924]
  MoveL 2529 to (-33.9, 37.89, 50.44) mm, rotated rx 180 ry 0 rz 180 deg; joints [-36.509, -22.936, 87.946, 60.285, 43.238, -51.924]
  Call Extruder(459.36942)
  MoveL 2530 to (-33.6, 37.71, 50.44) mm, rotated rx 180 ry 0 rz 180 deg; joints [-36.439, -22.918, 87.935, 60.229, 43.179, -51.888]
  MoveL 2531 to (-33.6, 37.71, 50.44) mm, rotated rx 180 ry 0 rz 180 deg; joints [-36.439, -22.918, 87.935, 60.229, 43.179, -51.888]
  Call Extruder(459.57597)
  MoveL 2532 to (-33.29, 37.54, 50.44) mm, rotated rx -180 ry 0 rz 180 deg; joints [-36.368, -22.9, 87.925, 60.172, 43.119, -51.851]
  MoveL 2533 to (-33.29, 37.54, 50.44) mm, rotated rx -180 ry 0 rz 180 deg; joints [-36.368, -22.9, 87.925, 60.172, 43.119, -51.851]
  Call Extruder(459.78174)
  MoveL 2534 to (-32.99, 37.36, 50.44) mm, rotated rx 180 ry 0 rz 180 deg; joints [-36.298, -22.881, 87.915, 60.116, 43.06, -51.815]
  MoveL 2535 to (-32.99, 37.36, 50.44) mm, rotated rx 180 ry 0 rz 180 deg; joints [-36.298, -22.881, 87.915, 60.116, 43.06, -51.815]
  Call Extruder(459.94004)
  MoveL 2536 to (-32.74, 37.26, 50.44) mm, rotated rx 180 ry 0 rz 180 deg; joints [-36.247, -22.864, 87.905, 60.077, 43.016, -51.791]
  MoveL 2537 to (-32.74, 37.26, 50.44) mm, rotated rx 180 ry 0 rz 180 deg; joints [-36.247, -22.864, 87.905, 60.077, 43.016, -51.791]
  Call Extruder(460.09774)
  MoveL 2538 to (-32.49, 37.15, 50.44) mm, rotated rx -180 ry 0 rz -180 deg; joints [-36.196, -22.846, 87.895, 60.038, 42.972, -51.767]
  MoveL 2539 to (-32.49, 37.15, 50.44) mm, rotated rx -180 ry 0 rz -180 deg; joints [-36.196, -22.846, 87.895, 60.038, 42.972, -51.767]
  Call Extruder(460.26783)
  MoveL 2540 to (-32.22, 37.04, 50.44) mm, rotated rx 180 ry 0 rz 180 deg; joints [-36.141, -22.827, 87.884, 59.996, 42.925, -51.741]
  MoveL 2541 to (-32.22, 37.04, 50.44) mm, rotated rx 180 ry 0 rz 180 deg; joints [-36.141, -22.827, 87.884, 59.996, 42.925, -51.741]
  Call Extruder(460.45016)
  MoveL 2542 to (-31.93, 36.91, 50.44) mm, rotated rx 180 ry 0 rz 180 deg; joints [-36.082, -22.805, 87.871, 59.951, 42.874, -51.713]
  MoveL 2543 to (-31.93, 36.91, 50.44) mm, rotated rx 180 ry 0 rz 180 deg; joints [-36.082, -22.805, 87.871, 59.951, 42.874, -51.713]
  Call Extruder(460.63174)
  MoveL 2544 to (-31.64, 36.79, 50.44) mm, rotated rx 180 ry 0 rz 180 deg; joints [-36.023, -22.784, 87.859, 59.906, 42.824, -51.685]
  MoveL 2545 to (-31.64, 36.79, 50.44) mm, rotated rx 180 ry 0 rz 180 deg; joints [-36.023, -22.784, 87.859, 59.906, 42.824, -51.685]
  Call Extruder(460.74519)
  MoveL 2546 to (-31.45, 36.73, 50.44) mm, rotated rx 180 ry 0 rz 180 deg; joints [-35.989, -22.769, 87.851, 59.88, 42.793, -51.67]
  MoveL 2547 to (-31.45, 36.73, 50.44) mm, rotated rx 180 ry 0 rz 180 deg; joints [-35.989, -22.769, 87.851, 59.88, 42.793, -51.67]
  Call Extruder(460.85821)
  MoveL 2548 to (-31.26, 36.67, 50.44) mm, rotated rx 180 ry 0 rz 180 deg; joints [-35.954, -22.754, 87.842, 59.854, 42.763, -51.655]
  MoveL 2549 to (-31.26, 36.67, 50.44) mm, rotated rx 180 ry 0 rz 180 deg; joints [-35.954, -22.754, 87.842, 59.854, 42.763, -51.655]
  Call Extruder(460.97078)
  MoveL 2550 to (-31.07, 36.61, 50.44) mm, rotated rx -180 ry 0 rz 180 deg; joints [-35.919, -22.739, 87.834, 59.828, 42.732, -51.64]
  MoveL 2551 to (-31.07, 36.61, 50.44) mm, rotated rx -180 ry 0 rz 180 deg; joints [-35.919, -22.739, 87.834, 59.828, 42.732, -51.64]
  Call Extruder(461.08290)
  MoveL 2552 to (-30.88, 36.55, 50.44) mm, rotated rx 180 ry 0 rz 180 deg; joints [-35.884, -22.724, 87.825, 59.802, 42.701, -51.625]
  MoveL 2553 to (-30.88, 36.55, 50.44) mm, rotated rx 180 ry 0 rz 180 deg; joints [-35.884, -22.724, 87.825, 59.802, 42.701, -51.625]
  Call Extruder(461.19458)
  MoveL 2554 to (-30.69, 36.49, 50.44) mm, rotated rx -180 ry 0 rz -180 deg; joints [-35.849, -22.709, 87.816, 59.777, 42.671, -51.609]
  MoveL 2555 to (-30.69, 36.49, 50.44) mm, rotated rx -180 ry 0 rz -180 deg; joints [-35.849, -22.709, 87.816, 59.777, 42.671, -51.609]
  Call Extruder(461.32566)
  MoveL 2556 to (-30.47, 36.42, 50.44) mm, rotated rx 180 ry 0 rz 180 deg; joints [-35.809, -22.691, 87.806, 59.747, 42.635, -51.592]
  MoveL 2557 to (-30.47, 36.42, 50.44) mm, rotated rx 180 ry 0 rz 180 deg; joints [-35.809, -22.691, 87.806, 59.747, 42.635, -51.592]
  Call Extruder(461.45616)
  MoveL 2558 to (-30.25, 36.35, 50.44) mm, rotated rx 180 ry 0 rz -180 deg; joints [-35.768, -22.672, 87.795, 59.717, 42.6, -51.575]
  MoveL 2559 to (-30.25, 36.35, 50.44) mm, rotated rx 180 ry 0 rz -180 deg; joints [-35.768, -22.672, 87.795, 59.717, 42.6, -51.575]
  Call Extruder(461.58611)
  MoveL 2560 to (-30.02, 36.28, 50.44) mm, rotated rx 180 ry 0 rz -180 deg; joints [-35.728, -22.654, 87.785, 59.688, 42.564, -51.558]
  MoveL 2561 to (-30.02, 36.28, 50.44) mm, rotated rx 180 ry 0 rz -180 deg; joints [-35.728, -22.654, 87.785, 59.688, 42.564, -51.558]
  Call Extruder(461.71549)
  MoveL 2562 to (-29.8, 36.22, 50.44) mm, rotated rx 180 ry 0 rz -180 deg; joints [-35.688, -22.636, 87.774, 59.658, 42.529, -51.54]
  MoveL 2563 to (-29.8, 36.22, 50.44) mm, rotated rx 180 ry 0 rz -180 deg; joints [-35.688, -22.636, 87.774, 59.658, 42.529, -51.54]
  Call Extruder(461.83745)
  MoveL 2564 to (-29.59, 36.16, 50.44) mm, rotated rx 180 ry 0 rz 180 deg; joints [-35.651, -22.618, 87.764, 59.631, 42.496, -51.525]
  MoveL 2565 to (-29.59, 36.16, 50.44) mm, rotated rx 180 ry 0 rz 180 deg; joints [-35.651, -22.618, 87.764, 59.631, 42.496, -51.525]
  Call Extruder(461.95230)
  MoveL 2566 to (-29.38, 36.12, 50.44) mm, rotated rx -180 ry 0 rz 180 deg; joints [-35.617, -22.599, 87.754, 59.607, 42.466, -51.512]
  MoveL 2567 to (-29.38, 36.12, 50.44) mm, rotated rx -180 ry 0 rz 180 deg; joints [-35.617, -22.599, 87.754, 59.607, 42.466, -51.512]
  Call Extruder(462.06669)
  MoveL 2568 to (-29.18, 36.07, 50.44) mm, rotated rx 180 ry 0 rz 180 deg; joints [-35.584, -22.581, 87.743, 59.584, 42.436, -51.499]
  MoveL 2569 to (-29.18, 36.07, 50.44) mm, rotated rx 180 ry 0 rz 180 deg; joints [-35.584, -22.581, 87.743, 59.584, 42.436, -51.499]
  Call Extruder(462.18063)
  MoveL 2570 to (-28.97, 36.03, 50.44) mm, rotated rx 180 ry 0 rz 180 deg; joints [-35.55, -22.563, 87.733, 59.56, 42.405, -51.486]
  MoveL 2571 to (-28.97, 36.03, 50.44) mm, rotated rx 180 ry 0 rz 180 deg; joints [-35.55, -22.563, 87.733, 59.56, 42.405, -51.486]
  Call Extruder(462.29412)
  MoveL 2572 to (-28.77, 35.98, 50.44) mm, rotated rx 180 ry 0 rz -180 deg; joints [-35.517, -22.545, 87.722, 59.536, 42.375, -51.473]
  MoveL 2573 to (-28.77, 35.98, 50.44) mm, rotated rx 180 ry 0 rz -180 deg; joints [-35.517, -22.545, 87.722, 59.536, 42.375, -51.473]
  Call Extruder(462.43141)
  MoveL 2574 to (-28.52, 35.93, 50.44) mm, rotated rx 180 ry 0 rz 180 deg; joints [-35.477, -22.523, 87.709, 59.508, 42.339, -51.458]
  MoveL 2575 to (-28.52, 35.93, 50.44) mm, rotated rx 180 ry 0 rz 180 deg; joints [-35.477, -22.523, 87.709, 59.508, 42.339, -51.458]
  Call Extruder(462.56808)
  MoveL 2576 to (-28.27, 35.88, 50.44) mm, rotated rx 180 ry 0 rz 180 deg; joints [-35.437, -22.5, 87.697, 59.48, 42.303, -51.443]
  MoveL 2577 to (-28.27, 35.88, 50.44) mm, rotated rx 180 ry 0 rz 180 deg; joints [-35.437, -22.5, 87.697, 59.48, 42.303, -51.443]
  Call Extruder(462.70414)
  MoveL 2578 to (-28.02, 35.83, 50.44) mm, rotated rx -180 ry 0 rz -180 deg; joints [-35.397, -22.478, 87.684, 59.452, 42.267, -51.427]
  MoveL 2579 to (-28.02, 35.83, 50.44) mm, rotated rx -180 ry 0 rz -180 deg; joints [-35.397, -22.478, 87.684, 59.452, 42.267, -51.427]
  Call Extruder(462.83959)
  MoveL 2580 to (-27.77, 35.78, 50.44) mm, rotated rx 180 ry 0 rz 180 deg; joints [-35.357, -22.455, 87.671, 59.424, 42.231, -51.412]
  MoveL 2581 to (-27.77, 35.78, 50.44) mm, rotated rx 180 ry 0 rz 180 deg; joints [-35.357, -22.455, 87.671, 59.424, 42.231, -51.412]
  Call Extruder(462.97443)
  MoveL 2582 to (-27.52, 35.73, 50.44) mm, rotated rx 180 ry 0 rz 180 deg; joints [-35.317, -22.433, 87.658, 59.396, 42.195, -51.397]
  MoveL 2583 to (-27.52, 35.73, 50.44) mm, rotated rx 180 ry 0 rz 180 deg; joints [-35.317, -22.433, 87.658, 59.396, 42.195, -51.397]
  Call Extruder(463.10867)
  MoveL 2584 to (-27.27, 35.68, 50.44) mm, rotated rx 180 ry 0 rz -180 deg; joints [-35.277, -22.41, 87.645, 59.368, 42.159, -51.382]
  MoveL 2585 to (-27.27, 35.68, 50.44) mm, rotated rx 180 ry 0 rz -180 deg; joints [-35.277, -22.41, 87.645, 59.368, 42.159, -51.382]
  Call Extruder(463.24229)
  MoveL 2586 to (-27.03, 35.64, 50.44) mm, rotated rx 180 ry 0 rz 180 deg; joints [-35.238, -22.388, 87.631, 59.341, 42.123, -51.367]
  MoveL 2587 to (-27.03, 35.64, 50.44) mm, rotated rx 180 ry 0 rz 180 deg; joints [-35.238, -22.388, 87.631, 59.341, 42.123, -51.367]
  Call Extruder(463.40438)
  MoveL 2588 to (-26.72, 35.59, 50.44) mm, rotated rx 180 ry 0 rz 180 deg; joints [-35.191, -22.359, 87.615, 59.309, 42.081, -51.35]
  MoveL 2589 to (-26.72, 35.59, 50.44) mm, rotated rx 180 ry 0 rz 180 deg; joints [-35.191, -22.359, 87.615, 59.309, 42.081, -51.35]
  Call Extruder(463.56576)
  MoveL 2590 to (-26.41, 35.54, 50.44) mm, rotated rx 180 ry 0 rz 180 deg; joints [-35.145, -22.33, 87.598, 59.277, 42.038, -51.334]
  MoveL 2591 to (-26.41, 35.54, 50.44) mm, rotated rx 180 ry 0 rz 180 deg; joints [-35.145, -22.33, 87.598, 59.277, 42.038, -51.334]
  Call Extruder(463.72640)
  MoveL 2592 to (-26.11, 35.49, 50.44) mm, rotated rx 180 ry 0 rz 180 deg; joints [-35.098, -22.301, 87.581, 59.245, 41.996, -51.317]
  MoveL 2593 to (-26.11, 35.49, 50.44) mm, rotated rx 180 ry 0 rz 180 deg; joints [-35.098, -22.301, 87.581, 59.245, 41.996, -51.317]
  Call Extruder(463.88631)
  MoveL 2594 to (-25.8, 35.44, 50.44) mm, rotated rx 180 ry 0 rz 180 deg; joints [-35.052, -22.273, 87.565, 59.214, 41.954, -51.3]
  MoveL 2595 to (-25.8, 35.44, 50.44) mm, rotated rx 180 ry 0 rz 180 deg; joints [-35.052, -22.273, 87.565, 59.214, 41.954, -51.3]
  Call Extruder(464.04550)
  MoveL 2596 to (-25.5, 35.39, 50.44) mm, rotated rx -180 ry 0 rz 180 deg; joints [-35.006, -22.244, 87.548, 59.182, 41.912, -51.284]
  MoveL 2597 to (-25.5, 35.39, 50.44) mm, rotated rx -180 ry 0 rz 180 deg; joints [-35.006, -22.244, 87.548, 59.182, 41.912, -51.284]
  Call Extruder(464.20396)
  MoveL 2598 to (-25.19, 35.34, 50.44) mm, rotated rx 180 ry 0 rz 180 deg; joints [-34.96, -22.215, 87.531, 59.15, 41.87, -51.267]
  MoveL 2599 to (-25.19, 35.34, 50.44) mm, rotated rx 180 ry 0 rz 180 deg; joints [-34.96, -22.215, 87.531, 59.15, 41.87, -51.267]
  Call Extruder(464.40284)
  MoveL 2600 to (-24.8, 35.3, 50.44) mm, rotated rx -180 ry 0 rz 180 deg; joints [-34.904, -22.177, 87.509, 59.113, 41.818, -51.248]
  MoveL 2601 to (-24.8, 35.3, 50.44) mm, rotated rx -180 ry 0 rz 180 deg; joints [-34.904, -22.177, 87.509, 59.113, 41.818, -51.248]
  Call Extruder(464.60085)
  MoveL 2602 to (-24.42, 35.25, 50.44) mm, rotated rx -180 ry 0 rz 180 deg; joints [-34.849, -22.14, 87.487, 59.076, 41.767, -51.23]
  MoveL 2603 to (-24.42, 35.25, 50.44) mm, rotated rx -180 ry 0 rz 180 deg; joints [-34.849, -22.14, 87.487, 59.076, 41.767, -51.23]
  Call Extruder(464.79799)
  MoveL 2604 to (-24.03, 35.21, 50.44) mm, rotated rx 180 ry 0 rz 180 deg; joints [-34.794, -22.102, 87.465, 59.039, 41.716, -51.211]
  MoveL 2605 to (-24.03, 35.21, 50.44) mm, rotated rx 180 ry 0 rz 180 deg; joints [-34.794, -22.102, 87.465, 59.039, 41.716, -51.211]
  Call Extruder(464.99426)
  MoveL 2606 to (-23.64, 35.16, 50.44) mm, rotated rx -180 ry 0 rz 180 deg; joints [-34.738, -22.064, 87.443, 59.002, 41.664, -51.193]
  MoveL 2607 to (-23.64, 35.16, 50.44) mm, rotated rx -180 ry 0 rz 180 deg; joints [-34.738, -22.064, 87.443, 59.002, 41.664, -51.193]
  Call Extruder(465.23995)
  MoveL 2608 to (-23.15, 35.11, 50.44) mm, rotated rx 180 ry 0 rz 180 deg; joints [-34.671, -22.015, 87.415, 58.958, 41.602, -51.171]
  MoveL 2609 to (-23.15, 35.11, 50.44) mm, rotated rx 180 ry 0 rz 180 deg; joints [-34.671, -22.015, 87.415, 58.958, 41.602, -51.171]
  Call Extruder(465.53467)
  MoveL 2610 to (-22.56, 35.07, 50.44) mm, rotated rx 180 ry 0 rz 180 deg; joints [-34.592, -21.956, 87.38, 58.907, 41.527, -51.147]
  MoveL 2611 to (-22.56, 35.07, 50.44) mm, rotated rx 180 ry 0 rz 180 deg; joints [-34.592, -21.956, 87.38, 58.907, 41.527, -51.147]
  Call Extruder(465.82807)
  MoveL 2612 to (-21.97, 35.02, 50.44) mm, rotated rx 180 ry 0 rz 180 deg; joints [-34.512, -21.896, 87.345, 58.856, 41.453, -51.122]
  MoveL 2613 to (-21.97, 35.02, 50.44) mm, rotated rx 180 ry 0 rz 180 deg; joints [-34.512, -21.896, 87.345, 58.856, 41.453, -51.122]
  Call Extruder(466.26140)
  MoveL 2614 to (-21.1, 34.98, 50.44) mm, rotated rx 180 ry 0 rz 180 deg; joints [-34.399, -21.806, 87.291, 58.784, 41.345, -51.089]
  MoveL 2615 to (-21.1, 34.98, 50.44) mm, rotated rx 180 ry 0 rz 180 deg; joints [-34.399, -21.806, 87.291, 58.784, 41.345, -51.089]
  Call Extruder(466.83356)
  MoveL 2616 to (-19.94, 34.93, 50.44) mm, rotated rx 180 ry 0 rz -180 deg; joints [-34.253, -21.685, 87.219, 58.693, 41.206, -51.049]
  MoveL 2617 to (-19.94, 34.93, 50.44) mm, rotated rx 180 ry 0 rz -180 deg; joints [-34.253, -21.685, 87.219, 58.693, 41.206, -51.049]
  Call Extruder(467.26139)
  MoveL 2618 to (-19.06, 34.91, 50.44) mm, rotated rx 180 ry 0 rz 180 deg; joints [-34.146, -21.592, 87.164, 58.628, 41.103, -51.021]
  Call Extruder(583.91008)
  MoveL 2619 to (219.06, 34.91, 50.44) mm, rotated rx 180 ry 0 rz 180 deg; joints [-18.248, 10.699, 58.135, 42.402, 27.67, -38.964]
  MoveL 2620 to (219.06, 34.91, 50.44) mm, rotated rx 180 ry 0 rz 180 deg; joints [-18.248, 10.699, 58.135, 42.402, 27.67, -38.964]
  Call Extruder(584.62565)
  MoveL 2621 to (220.52, 34.95, 50.44) mm, rotated rx -180 ry 0 rz 180 deg; joints [-18.199, 10.955, 57.829, 42.254, 27.676, -38.818]
  MoveL 2622 to (220.52, 34.95, 50.44) mm, rotated rx -180 ry 0 rz 180 deg; joints [-18.199, 10.955, 57.829, 42.254, 27.676, -38.818]
  Call Extruder(585.20039)
  MoveL 2623 to (221.68, 35, 50.44) mm, rotated rx 180 ry 0 rz 180 deg; joints [-18.162, 11.161, 57.581, 42.138, 27.684, -38.702]
  MoveL 2624 to (221.68, 35, 50.44) mm, rotated rx 180 ry 0 rz 180 deg; joints [-18.162, 11.161, 57.581, 42.138, 27.684, -38.702]
  Call Extruder(585.49378)
  MoveL 2625 to (222.27, 35.05, 50.44) mm, rotated rx 180 ry 0 rz 180 deg; joints [-18.146, 11.267, 57.453, 42.083, 27.69, -38.646]
  MoveL 2626 to (222.27, 35.05, 50.44) mm, rotated rx 180 ry 0 rz 180 deg; joints [-18.146, 11.267, 57.453, 42.083, 27.69, -38.646]
  Call Extruder(585.78851)
  MoveL 2627 to (222.86, 35.09, 50.44) mm, rotated rx -180 ry 0 rz -180 deg; joints [-18.13, 11.373, 57.325, 42.028, 27.696, -38.59]
  MoveL 2628 to (222.86, 35.09, 50.44) mm, rotated rx -180 ry 0 rz -180 deg; joints [-18.13, 11.373, 57.325, 42.028, 27.696, -38.59]
  Call Extruder(586.08457)
  MoveL 2629 to (223.45, 35.14, 50.44) mm, rotated rx 180 ry 0 rz 180 deg; joints [-18.113, 11.48, 57.196, 41.972, 27.703, -38.534]
  MoveL 2630 to (223.45, 35.14, 50.44) mm, rotated rx 180 ry 0 rz 180 deg; joints [-18.113, 11.48, 57.196, 41.972, 27.703, -38.534]
  Call Extruder(586.28084)
  MoveL 2631 to (223.84, 35.18, 50.44) mm, rotated rx 180 ry 0 rz -180 deg; joints [-18.104, 11.55, 57.11, 41.938, 27.708, -38.499]
  MoveL 2632 to (223.84, 35.18, 50.44) mm, rotated rx 180 ry 0 rz -180 deg; joints [-18.104, 11.55, 57.11, 41.938, 27.708, -38.499]
  Call Extruder(586.47798)
  MoveL 2633 to (224.22, 35.23, 50.44) mm, rotated rx 180 ry 0 rz 180 deg; joints [-18.095, 11.622, 57.024, 41.903, 27.714, -38.464]
  MoveL 2634 to (224.22, 35.23, 50.44) mm, rotated rx 180 ry 0 rz 180 deg; joints [-18.095, 11.622, 57.024, 41.903, 27.714, -38.464]
  Call Extruder(586.67599)
  MoveL 2635 to (224.61, 35.28, 50.44) mm, rotated rx 180 ry 0 rz 180 deg; joints [-18.087, 11.693, 56.937, 41.869, 27.72, -38.429]
  MoveL 2636 to (224.61, 35.28, 50.44) mm, rotated rx 180 ry 0 rz 180 deg; joints [-18.087, 11.693, 56.937, 41.869, 27.72, -38.429]
  Call Extruder(586.87487)
  MoveL 2637 to (225, 35.32, 50.44) mm, rotated rx -180 ry 0 rz 180 deg; joints [-18.078, 11.764, 56.851, 41.835, 27.726, -38.394]
  MoveL 2638 to (225, 35.32, 50.44) mm, rotated rx -180 ry 0 rz 180 deg; joints [-18.078, 11.764, 56.851, 41.835, 27.726, -38.394]
  Call Extruder(587.05395)
  MoveL 2639 to (225.34, 35.37, 50.44) mm, rotated rx -180 ry 0 rz 180 deg; joints [-18.07, 11.828, 56.773, 41.805, 27.732, -38.363]
  MoveL 2640 to (225.34, 35.37, 50.44) mm, rotated rx -180 ry 0 rz 180 deg; joints [-18.07, 11.828, 56.773, 41.805, 27.732, -38.363]
  Call Extruder(587.21313)
  MoveL 2641 to (225.65, 35.42, 50.44) mm, rotated rx 180 ry 0 rz 180 deg; joints [-18.065, 11.885, 56.703, 41.779, 27.737, -38.337]
  MoveL 2642 to (225.65, 35.42, 50.44) mm, rotated rx 180 ry 0 rz 180 deg; joints [-18.065, 11.885, 56.703, 41.779, 27.737, -38.337]
  Call Extruder(587.37304)
  MoveL 2643 to (225.96, 35.46, 50.44) mm, rotated rx 180 ry 0 rz 180 deg; joints [-18.059, 11.943, 56.633, 41.754, 27.743, -38.31]
  MoveL 2644 to (225.96, 35.46, 50.44) mm, rotated rx 180 ry 0 rz 180 deg; joints [-18.059, 11.943, 56.633, 41.754, 27.743, -38.31]
  Call Extruder(587.53368)
  MoveL 2645 to (226.26, 35.51, 50.44) mm, rotated rx 180 ry 0 rz 180 deg; joints [-18.054, 12, 56.564, 41.729, 27.749, -38.284]
  MoveL 2646 to (226.26, 35.51, 50.44) mm, rotated rx 180 ry 0 rz 180 deg; joints [-18.054, 12, 56.564, 41.729, 27.749, -38.284]
  Call Extruder(587.69505)
  MoveL 2647 to (226.57, 35.56, 50.44) mm, rotated rx -180 ry 0 rz -180 deg; joints [-18.048, 12.057, 56.494, 41.703, 27.755, -38.257]
  MoveL 2648 to (226.57, 35.56, 50.44) mm, rotated rx -180 ry 0 rz -180 deg; joints [-18.048, 12.057, 56.494, 41.703, 27.755, -38.257]
  Call Extruder(587.85714)
  MoveL 2649 to (226.87, 35.61, 50.44) mm, rotated rx 180 ry 0 rz 180 deg; joints [-18.042, 12.114, 56.423, 41.678, 27.761, -38.231]
  MoveL 2650 to (226.87, 35.61, 50.44) mm, rotated rx 180 ry 0 rz 180 deg; joints [-18.042, 12.114, 56.423, 41.678, 27.761, -38.231]
  Call Extruder(588.00405)
  MoveL 2651 to (227.15, 35.66, 50.44) mm, rotated rx 180 ry 0 rz -180 deg; joints [-18.038, 12.166, 56.36, 41.655, 27.767, -38.207]
  MoveL 2652 to (227.15, 35.66, 50.44) mm, rotated rx 180 ry 0 rz -180 deg; joints [-18.038, 12.166, 56.36, 41.655, 27.767, -38.207]
  Call Extruder(588.13568)
  MoveL 2653 to (227.39, 35.71, 50.44) mm, rotated rx 180 ry 0 rz 180 deg; joints [-18.034, 12.213, 56.303, 41.636, 27.773, -38.188]
  MoveL 2654 to (227.39, 35.71, 50.44) mm, rotated rx 180 ry 0 rz 180 deg; joints [-18.034, 12.213, 56.303, 41.636, 27.773, -38.188]
  Call Extruder(588.26790)
  MoveL 2655 to (227.64, 35.76, 50.44) mm, rotated rx 180 ry 0 rz -180 deg; joints [-18.031, 12.259, 56.246, 41.617, 27.778, -38.168]
  MoveL 2656 to (227.64, 35.76, 50.44) mm, rotated rx 180 ry 0 rz -180 deg; joints [-18.031, 12.259, 56.246, 41.617, 27.778, -38.168]
  Call Extruder(588.40071)
  MoveL 2657 to (227.88, 35.81, 50.44) mm, rotated rx -180 ry 0 rz 180 deg; joints [-18.028, 12.306, 56.189, 41.598, 27.784, -38.147]
  MoveL 2658 to (227.88, 35.81, 50.44) mm, rotated rx -180 ry 0 rz 180 deg; joints [-18.028, 12.306, 56.189, 41.598, 27.784, -38.147]
  Call Extruder(588.53410)
  MoveL 2659 to (228.12, 35.85, 50.44) mm, rotated rx 180 ry 0 rz -180 deg; joints [-18.024, 12.353, 56.132, 41.58, 27.79, -38.127]
  MoveL 2660 to (228.12, 35.85, 50.44) mm, rotated rx 180 ry 0 rz -180 deg; joints [-18.024, 12.353, 56.132, 41.58, 27.79, -38.127]
  Call Extruder(588.66808)
  MoveL 2661 to (228.37, 35.9, 50.44) mm, rotated rx -180 ry 0 rz 180 deg; joints [-18.021, 12.399, 56.075, 41.56, 27.796, -38.107]
  MoveL 2662 to (228.37, 35.9, 50.44) mm, rotated rx -180 ry 0 rz 180 deg; joints [-18.021, 12.399, 56.075, 41.56, 27.796, -38.107]
  Call Extruder(588.80265)
  MoveL 2663 to (228.61, 35.95, 50.44) mm, rotated rx 180 ry 0 rz -180 deg; joints [-18.017, 12.446, 56.017, 41.541, 27.802, -38.087]
  MoveL 2664 to (228.61, 35.95, 50.44) mm, rotated rx 180 ry 0 rz -180 deg; joints [-18.017, 12.446, 56.017, 41.541, 27.802, -38.087]
  Call Extruder(588.88871)
  MoveL 2665 to (228.77, 35.98, 50.44) mm, rotated rx -180 ry 0 rz 180 deg; joints [-18.015, 12.476, 55.981, 41.529, 27.805, -38.074]
  MoveL 2666 to (228.77, 35.98, 50.44) mm, rotated rx -180 ry 0 rz 180 deg; joints [-18.015, 12.476, 55.981, 41.529, 27.805, -38.074]
  Call Extruder(589.00224)
  MoveL 2667 to (228.97, 36.02, 50.44) mm, rotated rx -180 ry 0 rz 180 deg; joints [-18.012, 12.515, 55.932, 41.513, 27.81, -38.057]
  MoveL 2668 to (228.97, 36.02, 50.44) mm, rotated rx -180 ry 0 rz 180 deg; joints [-18.012, 12.515, 55.932, 41.513, 27.81, -38.057]
  Call Extruder(589.11625)
  MoveL 2669 to (229.18, 36.06, 50.44) mm, rotated rx -180 ry 0 rz -180 deg; joints [-18.009, 12.554, 55.884, 41.496, 27.815, -38.04]
  MoveL 2670 to (229.18, 36.06, 50.44) mm, rotated rx -180 ry 0 rz -180 deg; joints [-18.009, 12.554, 55.884, 41.496, 27.815, -38.04]
  Call Extruder(589.23074)
  MoveL 2671 to (229.38, 36.1, 50.44) mm, rotated rx -180 ry 0 rz 180 deg; joints [-18.006, 12.593, 55.836, 41.48, 27.82, -38.022]
  MoveL 2672 to (229.38, 36.1, 50.44) mm, rotated rx -180 ry 0 rz 180 deg; joints [-18.006, 12.593, 55.836, 41.48, 27.82, -38.022]
  Call Extruder(589.35620)
  MoveL 2673 to (229.6, 36.16, 50.44) mm, rotated rx 180 ry 0 rz 180 deg; joints [-18.006, 12.637, 55.782, 41.466, 27.827, -38.007]
  MoveL 2674 to (229.6, 36.16, 50.44) mm, rotated rx 180 ry 0 rz 180 deg; joints [-18.006, 12.637, 55.782, 41.466, 27.827, -38.007]
  Call Extruder(589.48218)
  MoveL 2675 to (229.82, 36.23, 50.44) mm, rotated rx 180 ry 0 rz 180 deg; joints [-18.005, 12.68, 55.729, 41.452, 27.834, -37.992]
  MoveL 2676 to (229.82, 36.23, 50.44) mm, rotated rx 180 ry 0 rz 180 deg; joints [-18.005, 12.68, 55.729, 41.452, 27.834, -37.992]
  Call Extruder(589.60868)
  MoveL 2677 to (230.04, 36.29, 50.44) mm, rotated rx 180 ry 0 rz 180 deg; joints [-18.004, 12.723, 55.676, 41.438, 27.842, -37.976]
  MoveL 2678 to (230.04, 36.29, 50.44) mm, rotated rx 180 ry 0 rz 180 deg; joints [-18.004, 12.723, 55.676, 41.438, 27.842, -37.976]
  Call Extruder(589.73571)
  MoveL 2679 to (230.26, 36.36, 50.44) mm, rotated rx 180 ry 0 rz 180 deg; joints [-18.003, 12.766, 55.622, 41.424, 27.849, -37.961]
  MoveL 2680 to (230.26, 36.36, 50.44) mm, rotated rx 180 ry 0 rz 180 deg; joints [-18.003, 12.766, 55.622, 41.424, 27.849, -37.961]
  Call Extruder(589.86325)
  MoveL 2681 to (230.48, 36.42, 50.44) mm, rotated rx 180 ry 0 rz -180 deg; joints [-18.003, 12.809, 55.569, 41.411, 27.856, -37.945]
  MoveL 2682 to (230.48, 36.42, 50.44) mm, rotated rx 180 ry 0 rz -180 deg; joints [-18.003, 12.809, 55.569, 41.411, 27.856, -37.945]
  Call Extruder(589.99132)
  MoveL 2683 to (230.69, 36.49, 50.44) mm, rotated rx 180 ry 0 rz 180 deg; joints [-18.002, 12.853, 55.515, 41.397, 27.863, -37.93]
  MoveL 2684 to (230.69, 36.49, 50.44) mm, rotated rx 180 ry 0 rz 180 deg; joints [-18.002, 12.853, 55.515, 41.397, 27.863, -37.93]
  Call Extruder(590.10322)
  MoveL 2685 to (230.88, 36.55, 50.44) mm, rotated rx 180 ry 0 rz 180 deg; joints [-18.002, 12.891, 55.469, 41.385, 27.87, -37.917]
  MoveL 2686 to (230.88, 36.55, 50.44) mm, rotated rx 180 ry 0 rz 180 deg; joints [-18.002, 12.891, 55.469, 41.385, 27.87, -37.917]
  Call Extruder(590.21556)
  MoveL 2687 to (231.07, 36.61, 50.44) mm, rotated rx -180 ry 0 rz 180 deg; joints [-18.002, 12.928, 55.422, 41.374, 27.877, -37.904]
  MoveL 2688 to (231.07, 36.61, 50.44) mm, rotated rx -180 ry 0 rz 180 deg; joints [-18.002, 12.928, 55.422, 41.374, 27.877, -37.904]
  Call Extruder(590.32835)
  MoveL 2689 to (231.26, 36.67, 50.44) mm, rotated rx 180 ry 0 rz 180 deg; joints [-18.002, 12.966, 55.375, 41.363, 27.883, -37.892]
  MoveL 2690 to (231.26, 36.67, 50.44) mm, rotated rx 180 ry 0 rz 180 deg; joints [-18.002, 12.966, 55.375, 41.363, 27.883, -37.892]
  Call Extruder(590.44158)
  MoveL 2691 to (231.45, 36.73, 50.44) mm, rotated rx -180 ry 0 rz -180 deg; joints [-18.002, 13.004, 55.328, 41.352, 27.89, -37.879]
  MoveL 2692 to (231.45, 36.73, 50.44) mm, rotated rx -180 ry 0 rz -180 deg; joints [-18.002, 13.004, 55.328, 41.352, 27.89, -37.879]
  Call Extruder(590.55526)
  MoveL 2693 to (231.64, 36.79, 50.44) mm, rotated rx -180 ry 0 rz 180 deg; joints [-18.002, 13.042, 55.281, 41.34, 27.897, -37.866]
  MoveL 2694 to (231.64, 36.79, 50.44) mm, rotated rx -180 ry 0 rz 180 deg; joints [-18.002, 13.042, 55.281, 41.34, 27.897, -37.866]
  Call Extruder(590.73722)
  MoveL 2695 to (231.93, 36.91, 50.44) mm, rotated rx -180 ry 0 rz 180 deg; joints [-18.005, 13.102, 55.206, 41.327, 27.91, -37.85]
  MoveL 2696 to (231.93, 36.91, 50.44) mm, rotated rx -180 ry 0 rz 180 deg; joints [-18.005, 13.102, 55.206, 41.327, 27.91, -37.85]
  Call Extruder(590.91994)
  MoveL 2697 to (232.22, 37.04, 50.44) mm, rotated rx -180 ry 0 rz -180 deg; joints [-18.008, 13.163, 55.131, 41.314, 27.922, -37.833]
  MoveL 2698 to (232.22, 37.04, 50.44) mm, rotated rx -180 ry 0 rz -180 deg; joints [-18.008, 13.163, 55.131, 41.314, 27.922, -37.833]
  Call Extruder(591.09035)
  MoveL 2699 to (232.49, 37.15, 50.44) mm, rotated rx -180 ry 0 rz 180 deg; joints [-18.011, 13.219, 55.062, 41.301, 27.934, -37.819]
  MoveL 2700 to (232.49, 37.15, 50.44) mm, rotated rx -180 ry 0 rz 180 deg; joints [-18.011, 13.219, 55.062, 41.301, 27.934, -37.819]
  Call Extruder(591.24835)
  MoveL 2701 to (232.74, 37.26, 50.44) mm, rotated rx 180 ry 0 rz -180 deg; joints [-18.013, 13.271, 54.997, 41.29, 27.946, -37.805]
  MoveL 2702 to (232.74, 37.26, 50.44) mm, rotated rx 180 ry 0 rz -180 deg; joints [-18.013, 13.271, 54.997, 41.29, 27.946, -37.805]
  Call Extruder(591.40695)
  MoveL 2703 to (232.99, 37.36, 50.44) mm, rotated rx 180 ry 0 rz 180 deg; joints [-18.016, 13.323, 54.933, 41.279, 27.957, -37.791]
  MoveL 2704 to (232.99, 37.36, 50.44) mm, rotated rx 180 ry 0 rz 180 deg; joints [-18.016, 13.323, 54.933, 41.279, 27.957, -37.791]
  Call Extruder(591.61312)
  MoveL 2705 to (233.29, 37.54, 50.44) mm, rotated rx 180 ry 0 rz 180 deg; joints [-18.024, 13.389, 54.85, 41.273, 27.974, -37.781]
  MoveL 2706 to (233.29, 37.54, 50.44) mm, rotated rx 180 ry 0 rz 180 deg; joints [-18.024, 13.389, 54.85, 41.273, 27.974, -37.781]
